# B&R Automation Studio project RS15_RX_30005_r00 (part 2)

#### A7_BasicCyclic.st - Cyclic code
```iecst
(********************************************************************
 * COPYRIGHT -- Microsoft
 ********************************************************************
 * Program: A7_Basic
 * File: A7_BasicCyclic.st
 * Author: pkiel
 * Created: July 13, 2011
 ********************************************************************
 * Implementation of program A7_Basic
 ********************************************************************)

PROGRAM _CYCLIC

	gA[7].UnitsPerInch := gA[7].AxisPeriod/gRecipeActive.Repeat;
  gA[7].InchPerDeg := gA[7].UnitsPerDeg / gA[7].UnitsPerInch ;
  IF (g_rNumbPliers <> 0.0) THEN
    gA[7].rPerim_In := g_rSizeDrum_mm/g_rNumbPliers/25.4 ;
    gA[7].rRSynNum := 4.0 / g_rNumbPliers ;
  END_IF ;
  gA[7].rRSynDen := 1.0 ;

	IF (gA[7].Ident<>0) THEN

	(************************ READ DRIVE STATUS *************************)
	(* Access to the following bools:
	gA[x]_DriveStatus.Simulation			: If TRUE, simulation mode is active
	gA[x]_DriveStatus.NetworkInit			: If TRUE, the network is initialized
	gA[x]_DriveStatus.HomeSwitch			: If TRUE, the digital reference switch input is active
	gA[x]_DriveStatus.PosHWSwitch			: If TRUE, the positive hardware end switch is active
	gA[x]_DriveStatus.NegHWSwitch			: If TRUE, the negative hardware end switch is active
	gA[x]_DriveStatus.Trigger1				: If TRUE, the first trigger input is active
	gA[x]_DriveStatus.Trigger2				: If TRUE, the second trigger input is active
	gA[x]_DriveStatus.DriveEnable			: If TRUE, the enable input is active
	gA[x]_DriveStatus.ControllerReady		: If TRUE, the controller is ready to beturned on
	gA[x]_DriveStatus.ControllerStatus		: If TRUE, the controller is turned on (Same as MC_Power.Status)
	gA[x]_DriveStatus.AxisError				: If TRUE, at least one error has occurred (not acknowledged)
	gA[x]_DriveStatus.LagWarning			: If TRUE, the lag error has exceeded the limit value specified for a warning*)
		MC_BR_ReadDriveStatus_0.Enable := 1;
		MC_BR_ReadDriveStatus_0.Axis := gA[7].Ident;
		MC_BR_ReadDriveStatus_0.AdrDriveStatus := ADR (DriveStatus);
		MC_BR_ReadDriveStatus_0();
		gA[7].Ind_Simulation		:=	DriveStatus.Simulation;
		gA[7].Ind_NetworkInit		:=	DriveStatus.NetworkInit;
		gA[7].Input_Home			:=	DriveStatus.HomeSwitch;
		gA[7].Input_PosHW			:=	DriveStatus.PosHWSwitch;
		gA[7].Input_NegHW			:=	DriveStatus.NegHWSwitch;
		gA[7].Input_Trigger1		:=	DriveStatus.Trigger1;
		gA[7].Input_Trigger2		:=	DriveStatus.Trigger2;
		gA[7].Input_DriveEnable		:=	DriveStatus.DriveEnable;
		gA[7].Ind_ControllerReady	:=	DriveStatus.ControllerReady;
		gA[7].Ind_ControllerStatus	:=	DriveStatus.ControllerStatus;
		gA[7].Error					:=	DriveStatus.AxisError;
		gA[7].Ind_LagWarning		:=	DriveStatus.LagWarning;

	(************************ READ AXIS ERROR **********************)
		MC_ReadAxisError_0.Enable := gA[7].Ind_NetworkInit;
		MC_ReadAxisError_0.Axis := gA[7].Ident;
		MC_ReadAxisError_0.DataAddress := ADR(gA[7].ErrorText);
		MC_ReadAxisError_0.DataLength := SIZEOF(gA[7].ErrorText);
		MC_ReadAxisError_0.DataObjectName := 'Error_Eng';
		MC_ReadAxisError_0();
		IF(MC_ReadAxisError_0.Valid) THEN
			gA[7].ErrorID := MC_ReadAxisError_0.AxisErrorID;
			gA[7].ErrorCount := MC_ReadAxisError_0.AxisErrorCount;
		END_IF
	(* Auto Acknowledge Errors *)
		IF (gA[7].Cmd_Reset AND (gA[7].ErrorCount<>0) AND NOT AutoAck) THEN
			AutoAck:=1;
		ELSE
			AutoAck:=0;
		END_IF
	(*Axis Error Acknowledge*)
		IF (EDGEPOS(AutoAck) OR EDGEPOS(gA[7].ErrorAck)) THEN
			MC_ReadAxisError_0.Acknowledge := 1;
		ELSE;
			MC_ReadAxisError_0.Acknowledge :=0;
		END_IF

	(************************ RESET AXIS ERROR **********************)
		IF (gA[7].Cmd_Reset AND (gA[7].ErrorCount=0) AND gA[7].ErrorStop) THEN
			MC_Reset_0.Execute:=1;
		END_IF
		IF (MC_Reset_0.Done) THEN
			MC_Reset_0.Execute:=0;
			gA[7].Cmd_Reset:=0;
			ResetError := 0;
		END_IF
		IF (MC_Reset_0.Error) THEN
			MC_Reset_0.Execute:=0;
			gA[7].Cmd_Reset:=0;
			ResetError := 1;
		END_IF
		MC_Reset_0.Axis:=gA[7].Ident;
		MC_Reset_0();

	(************************ READ AXIS STATUS *************************)
		MC_ReadStatus_0.Enable := gA[7].Ind_NetworkInit;
		MC_ReadStatus_0.Axis := gA[7].Ident;
		MC_ReadStatus_0();
		IF(MC_ReadStatus_0.Valid = TRUE)THEN
			gA[7].Ind_Enabled 			:= NOT (MC_ReadStatus_0.Disabled);
			gA[7].Ind_StandStill		:= MC_ReadStatus_0.StandStill;
			gA[7].Ind_Stopping			:= MC_ReadStatus_0.Stopping;
			gA[7].Ind_DiscreteMotion	:= MC_ReadStatus_0.DiscreteMotion;
			gA[7].Ind_ContinuousMotion	:= MC_ReadStatus_0.ContinuousMotion;
			gA[7].Ind_SynchronizedMotion:= MC_ReadStatus_0.SynchronizedMotion;
			gA[7].ErrorStop				:= MC_ReadStatus_0.Errorstop;
		END_IF
    IF NOT(gA[7].Ind_Enabled) THEN
      gA[7].bSynchroReq := 1 ;
    END_IF
    IF EDGEPOS(gA[7].Ind_bSynchroOK) THEN
      gA[7].bSynchroReq := 0 ;
    END_IF

	(******************** INIT POSITION MODULUS  *********************)
    IF (g_rNumbPliers <> 0.0) THEN
      IF ( gA[7].Ind_StandStill     OR
           NOT(gA[7].Ind_Enabled) ) AND
         g_bChangeModDrumReq        THEN
        bChangeModReq := 1 ;
        uiInitModPos0_ErrorID := 0 ;
      END_IF
      MC_BR_InitModPos_0.Execute:= (InitModPosition OR bChangeModReq) ;
  		MC_BR_InitModPos_0.Axis:= gA[7].Ident;
  		MC_BR_InitModPos_0.Period:= REAL_TO_UDINT(gA[7].AxisPeriod * 4.0/g_rNumbPliers);
  		MC_BR_InitModPos_0.Factor:=1;
  		InitModPos_Done:=MC_BR_InitModPos_0.Done;
    END_IF
    IF MC_BR_InitModPos_0.Done THEN
      g_bChangeModDrumReq := 0 ;
      bChangeModReq       := 0 ;
    ELSIF MC_BR_InitModPos_0.Error THEN
      bChangeModReq := 0 ;
      uiInitModPos0_ErrorID := MC_BR_InitModPos_0.ErrorID ;
    END_IF
		MC_BR_InitModPos_0();

	(******************** INIT ENDLESS POSITION *********************)
		MC_BR_InitEndlessPosition_0.Execute:= InitModPos_Done;
		MC_BR_InitEndlessPosition_0.Axis:= gA[7].Ident;
		MC_BR_InitEndlessPosition_0.DataAddress:= ADR(gEndPosData[7]);
		IF (MC_BR_InitEndlessPosition_0.Done) THEN
			InitModPosition:=0;
			InitEndlessPosition:=0;
			HomeRestore:=1;
		END_IF
		MC_BR_InitEndlessPosition_0();

	(************************ HOME AXIS FIRST POWER UP **********************)
		IF (HomeRestore AND NOT gA7_FirstHomed) THEN
			MC_Home_0.Execute:=1;
		END_IF
		MC_Home_0.Axis:=gA[7].Ident;
		MC_Home_0.Position:=0;
		MC_Home_0.HomingMode:=mcHOME_DIRECT;
		IF (MC_Home_0.Done) THEN
			MC_Home_0.Execute:=0;
			gA7_FirstHomed:=1;
		END_IF
		MC_Home_0();

	(************************ HOME AXIS **********************)
		IF (gA7_FirstHomed) THEN
			MC_Home_1.Execute:=HomeRestore;
		END_IF
		MC_Home_1.Axis:=gA[7].Ident;
		MC_Home_1.Position:=0;
		MC_Home_1.HomingMode:=mcHOME_RESTORE_POS;
		IF (MC_Home_1.Done) THEN
			gA[7].Ind_Homed:=1;
			HomeRestore:=0;
		END_IF
		MC_Home_1();

	(******************** READ ACTUAL POSITION *********************)
		MC_ReadActualPosition_0.Enable:= gA[7].Ind_NetworkInit;
		MC_ReadActualPosition_0.Axis:= gA[7].Ident;
		MC_ReadActualPosition_0();
		IF(MC_ReadActualPosition_0.Valid = TRUE)THEN
			gA[7].PositionCount := MC_ReadActualPosition_0.Position;
			gA[7].PositionInch := gA[7].PositionCount/gA[7].UnitsPerInch;
			gA[7].PositionDeg := gA[7].PositionCount/gA[7].UnitsPerDeg;
		END_IF

  //******************** READ SET POINT POSITION *********************
    // Slave side  : ParID 428 SGEN_S_SET : CTRL Position controller: Input set position
    // Master side : ParID 412 S_SET_VAX1 : 412: VAX: Position

    // Slave side
    MC_BR_CyclicRead_0.Axis        := gA[7].Ident ;
    MC_BR_CyclicRead_0.Enable      := gA[7].Ind_NetworkInit;
    MC_BR_CyclicRead_0.ParID       := 428 ;
    MC_BR_CyclicRead_0.DataAddress := ADR(iiSP_SlPos_U);
    MC_BR_CyclicRead_0.DataType    := ncPAR_TYP_DINT ;
    // Master side
    MC_BR_CyclicRead_1.Axis        := gA[9].Ident ;
    MC_BR_CyclicRead_1.Enable      := gA[7].Ind_NetworkInit;
    MC_BR_CyclicRead_1.ParID       := 412 ;
    MC_BR_CyclicRead_1.DataAddress := ADR(iiSP_MaPos_U);
    MC_BR_CyclicRead_1.DataType    := ncPAR_TYP_DINT ;

    IF MC_BR_CyclicRead_0.Valid THEN
      rSP_SlPos_Deg := iiSP_SlPos_U/gA[7].UnitsPerDeg ;
    ELSIF MC_BR_CyclicRead_0.Error THEN
      MC_BR_CyclicRead_0.Enable := 0 ;
    END_IF
    IF MC_BR_CyclicRead_1.Valid THEN
      rSP_MaPos_Deg := iiSP_MaPos_U/gA[9].UnitsPerDeg ;
    ELSIF MC_BR_CyclicRead_1.Error THEN
      MC_BR_CyclicRead_1.Enable := 0 ;
    END_IF
    MC_BR_CyclicRead_0();
    MC_BR_CyclicRead_1();

  //******************** READ ACTUAL OFFSET *********************
  IF gA[7].rRSynDen > 0.0 THEN
    rTempActPhasDeg := rSP_SlPos_Deg - gA[7].rRSynNum / gA[7].rRSynDen * rSP_MaPos_Deg ;
    gA[7].rActPhasDeg := H_FC_Modulus (
                              IN_rMod := 360 * gA[7].rRSynNum / gA[7].rRSynDen ,
                              IN_rVar := rTempActPhasDeg
                                      ) ;
  END_IF

	(******************** READ ACTUAL VELOCITY *********************)
		IF(MC_ReadActualVelocity_0.Error=TRUE) THEN
			MC_ReadActualVelocity_0.Enable:= 0;
		ELSE
			MC_ReadActualVelocity_0.Enable:= 1;
		END_IF
		MC_ReadActualVelocity_0.Axis:= gA[7].Ident;
		MC_ReadActualVelocity_0();
		IF(MC_ReadActualVelocity_0.Valid = TRUE)THEN
			//gA[7].ActualVelocity := MC_ReadActualVelocity_0.Velocity*60/gA[7].SP_MotorPPR;
      gA[7].ActualVelocity := MC_ReadActualVelocity_0.Velocity*60/gA[7].AxisPeriod ; // D.M. 03/08/2011 BrownPaper_14542  Need speed of the axis and not of the shaft of the motor
      IF ABS(gA[7].ActualVelocity>1) THEN // D.M. 03/08/2011 BrownPaper_14542 Add ABS because in case negative velocity Ind_InMotion = 0 instead of 1
				gA[7].Ind_InMotion:=1;
			ELSE
				gA[7].Ind_InMotion:=0;
			END_IF
		END_IF

	(******************** READ ACTUAL TORQUE *********************)
		IF(MC_ReadActualTorque_0.Error=TRUE) THEN
			MC_ReadActualTorque_0.Enable:= 0;
		ELSE
			MC_ReadActualTorque_0.Enable:= 1;
		END_IF
		MC_ReadActualTorque_0.Axis:= gA[7].Ident;
		MC_ReadActualTorque_0();
		IF(MC_ReadActualTorque_0.Valid = TRUE)THEN
			gA[7].ActualTorque := MC_ReadActualTorque_0.Torque;
		END_IF

	(************************ ENABLE AXIS **********************)
		MC_Power_0.Axis:=gA[7].Ident;
		IF (MC_Power_0.Error=0) THEN
			MC_Power_0.Enable:=gA[7].Cmd_Enable;
		ELSE;
			MC_Power_0.Enable:=0;
		END_IF;
		MC_Power_0();

	(************************ AXIS VELOCITY MOVE **********************)
		MC_MoveVelocity_0.Axis:=gA[7].Ident;
		MC_MoveVelocity_0.Velocity:=gA[7].SP_Velocity*gA[7].AxisPeriod/60;
		MC_MoveVelocity_0.Acceleration:=gA[7].SP_Accel;
		MC_MoveVelocity_0.Deceleration:=gA[7].SP_Decel;
		MC_MoveVelocity_0.Direction:=mcPOSITIVE_DIR;
		IF ((EDGEPOS(gA[7].Cmd_ContinuousMotion)) OR (EDGEPOS(gA[7].Cmd_ContinuousMotionUpdate))) THEN
			MC_MoveVelocity_0.Execute:=1;
		ELSE
			MC_MoveVelocity_0.Execute:=0;
		END_IF;
		MC_MoveVelocity_0();

  //************************ AXIS OVERRIDE **********************
    MC_SetOverride_0.Axis      := gA[7].Ident ;
    MC_SetOverride_0.Enable    := gA[7].Cmd_Override ;
    MC_SetOverride_0.VelFactor := gA[7].rSP_OverrideV ;
    MC_SetOverride_0.AccFactor := gA[7].rSP_OverrideA ;
    IF (MC_SetOverride_0.Enabled) OR
       (MC_SetOverride_0.Error)   THEN
      gA[7].Cmd_Override := 0 ;
    END_IF
    MC_SetOverride_0();

	(************************ AXIS STOP **********************)
		MC_Stop_0.Axis:=gA[7].Ident;
		IF (gA[7].Ind_ContinuousMotion AND (NOT gA[7].Cmd_ContinuousMotion) AND gAlarmsOK) THEN
			MC_Stop_0.Deceleration:=gA[7].SP_Decel;
			MC_Stop_0.Execute:=1;
		END_IF;
		IF (MC_Stop_0.Done OR MC_Stop_0.CommandAborted OR MC_Stop_0.Error) THEN
			MC_Stop_0.Execute:=0;
		END_IF;
		MC_Stop_0();

  (************************  ESTOP **********************)
    MC_Stop_1.Axis:=gA[7].Ident;
    IF EDGEPOS(g_bIndEStopStandstill) THEN
      MC_Stop_1.Deceleration:=gA[7].SP_EStopDecel;
      MC_Stop_1.Execute:=1;
    END_IF;
    IF (MC_Stop_1.Done OR MC_Stop_1.CommandAborted OR MC_Stop_1.Error) THEN
      MC_Stop_1.Execute:=0;
      gA[7].Cmd_EStopDisable := 1 ;
    END_IF;
    IF NOT(g_bIndEStopStandstill) THEN
      gA[7].Cmd_EStopDisable := 0 ;
    END_IF;
    MC_Stop_1();

    //************************ AXIS PHASE CONTROL (Inches) First Step **********************
    IF EDGEPOS(gA[7].Cmd_PhaseOffset) THEN
      rSP_PhaseOffsetVal := gA[7].SP_PhaseOffset ;
    END_IF;

    (************************ SHIFTING PERF CONTROL **********************)
    IF g_bCmdShiftA[7] THEN
      //rSP_ShiftDrum := g_iPerfShiftPos * gr_rIncrShiftPerf_mm/25.4 * gA[7].rRSynNum/gA[7].rRSynDen ;  // D.M. RS26_Pyrollpack_14661 CAUTION !!! Phasing acts on the master side and not slave side, replaced by the code below
      rSP_ShiftDrum := g_iPerfShiftPos * gr_rIncrShiftPerf_mm/25.4 ;
      gA[7].Cmd_PhaseOffset := 1 ;
      g_bCmdShiftA[7] := 0 ;
    END_IF

    (************************ AXIS PHASE CONTROL (Inches) Next Step **********************)
    // The biggers Offsets are divided in several successives shifts to not damage the blades on the Drum du to too much acceleration
    IF gA[7].Cmd_PhaseOffset               AND
       ( EDGENEG(gA[7].Ind_bInContactZone) AND
         (g_iMachType <> C_iRS15)          OR
         EDGENEG(gA[4].Ind_bInContactZone) AND
         (g_iMachType = C_iRS15) )         THEN
      gA[7].Cmd_PhaseOffset := 0 ;
      rSP_PhaseOffset := rSP_PhaseOffsetVal + rSP_ShiftDrum ;
      bCmd_PhaseOffset := 1 ;
      g_bIndPhasDrumInact := 0 ;
      //iTest_[0] := 0 ;
      //iTest_[1] := 0 ;
      //iTest_[2] := 0 ;
      //iTest_[3] := 0 ;
    END_IF
    rMaxShift := gr_rLimOffsetRunVal * gRecipeActive.Repeat ;
    // Signe of the Offset
    IF (rSP_PhaseOffset <> 0.0) THEN
      rShiftSign := rSP_PhaseOffset / ABS(rSP_PhaseOffset) ;
    END_IF
    // Shift calculation
    IF bCmd_PhaseOffset THEN
      IF (ABS(rSP_PhaseOffset) > rMaxShift) THEN
        rSP_ShiftVal := rMaxShift * rShiftSign ;
        rSP_PhaseOffset := rSP_PhaseOffset - rSP_ShiftVal ;
        iTest_[0] := iTest_[0] + 1 ;
      ELSE
        rSP_ShiftVal := rSP_PhaseOffset ;
        rSP_PhaseOffset := 0.0 ;
        iTest_[1] := iTest_[1] + 1 ;
      END_IF
    END_IF

    MC_BR_Phasing_0.Slave:=gA[7].Ident;
    IF gA[7].Ind_SynchronizedMotion AND NOT(gstCycA[7].CycManTimSet.bSCyc) AND st_TON_0.Q THEN
      MC_BR_Phasing_0.Enable:= 1;
    ELSE;
      MC_BR_Phasing_0.Enable:=0;
    END_IF;
    IF bCmd_PhaseOffset AND NOT(gstCycA[7].CycManTimSet.bSCyc) THEN
      MC_BR_Phasing_0.InitData:=1;
      bCmd_PhaseOffset := 0 ;
      IF (rSP_PhaseOffset = 0.0) THEN
        // Calculation new phase Drum/Master
        rTemp_[4] := (rSP_PhaseOffsetVal+rSP_ShiftDrum)/gA[7].InchPerDeg ;
        rTemp_[5] := gRecipeActive.rDrum_PhasMasterDeg + rTemp_[4]*gA[7].rRSynNum/gA[7].rRSynDen ;
        gRecipeActive.rDrum_PhasMasterDeg := H_FC_Modulus (IN_rMod := 360*gA[7].rRSynNum/gA[7].rRSynDen, IN_rVar := rTemp_[5]) ;
        rSP_ShiftDrum := 0.0 ;
        rSP_PhaseOffsetVal := 0 ;
        iTest_[2] := iTest_[2] + 1 ;
      END_IF;
    ELSE
      MC_BR_Phasing_0.InitData:=0;
    END_IF
    MC_BR_Phasing_0.Shift               := rSP_ShiftVal*gA[9].UnitsPerInch;
    MC_BR_Phasing_0.Velocity            := 6*gA[7].AxisPeriod/60;
    MC_BR_Phasing_0.Acceleration        := gA[7].SP_Decel;
    MC_BR_Phasing_0.ApplicationDistance := 0.8*gA[9].AxisPeriod * gA[7].rRSynNum/gA[7].rRSynDen ;
    MC_BR_Phasing_0.ApplicationMode     := mcMASTER_DISTANCE_BASED;
    MC_BR_Phasing_0.ShiftMode           := mcRELATIVE;
    MC_BR_Phasing_0();

    IF MC_BR_Phasing_0.ShiftAttained       AND
       (rSP_PhaseOffset <> 0.0)            AND
       ( EDGENEG(gA[7].Ind_bInContactZone) AND
         (g_iMachType <> C_iRS15)          OR
         EDGENEG(gA[4].Ind_bInContactZone) AND
         (g_iMachType = C_iRS15) )         THEN
      bCmd_PhaseOffset := 1 ;
      iTest_[3] := iTest_[3] + 1 ;
    END_IF
    // Drum phasing inactive
    IF (rSP_PhaseOffset=0.0)         AND
       MC_BR_Phasing_0.ShiftAttained OR
       NOT(MC_BR_Phasing_0.Busy)     AND
       1                             THEN
      g_bIndPhasDrumInact := 1 ;
    END_IF

    (************************ AXIS PHASE CONTROL (Inches) TIMING SETTING **********************)
    IF gstCycA[7].CycManTimSet.bSCyc THEN
      IF gA[7].Cmd_ManuTimSetPlus THEN
        rAxisTimSet_SP_Vel := gr_rAxisTimSet_SP_Vel*gA[9].AxisPeriod/60 / (gA[7].rRSynNum/gA[7].rRSynDen) ;
      ELSE
        rAxisTimSet_SP_Vel := - gr_rAxisTimSet_SP_Vel*gA[9].AxisPeriod/60 / (gA[7].rRSynNum/gA[7].rRSynDen) ;
      END_IF
        rAxisTimSet_SP_Acc := gr_rAxisTimSet_SP_Acc*gA[9].AxisPeriod/60/60 ;
    END_IF

    MC_BR_Phasing_1.Slave                  := gA[7].Ident;
    MC_BR_Phasing_1.Enable                 := gstCycA[7].CycManTimSet.bCyc ;
    MC_BR_Phasing_1.InitData               := gstCycA[7].CycManTimSet.bSCyc ;
    MC_BR_Phasing_1.PerformVelocityControl := gstCycA[7].CycManTimSet.CmdMov ;
    MC_BR_Phasing_1.Velocity               := rAxisTimSet_SP_Vel ;
    MC_BR_Phasing_1.Acceleration           := rAxisTimSet_SP_Acc ;
    MC_BR_Phasing_1.ApplicationMode        := mcVELOCITY_CONTROL ;
    MC_BR_Phasing_1();
    st_TON_0(IN:=NOT(MC_BR_Phasing_1.Enable),PT:=T#100ms) ;

    IF NOT(gstCycA[7].CycManTimSet.CmdMov) AND
       MC_BR_Phasing_1.ShiftAttained       OR
       NOT(gstCycA[7].CycManTimSet.bCyc)   OR
       MC_BR_Phasing_1.Error               AND
       1                                   THEN
      gstCycA[7].CycManTimSet.CmdStop := 0 ;
    END_IF
	END_IF

END_PROGRAM
```

#### A7_Basic.var - Local variables
```iecst
(********************************************************************
 * COPYRIGHT -- Microsoft
 ********************************************************************
 * Program: A7_Basic
 * File: A7_Basic.var
 * Author: pkiel
 * Created: July 13, 2011
 ********************************************************************
 * Local variables of program A7_Basic
 ********************************************************************)
VAR
	AutoAck : BOOL;
	AxisErrorNcAccess : UINT;
	DriveStatus : MC_DRIVESTATUS_TYP;
	HomeRestore : BOOL;
	InitEndlessPosition : BOOL;
	InitModPos_Done : BOOL;
	InitModPosition : BOOL;
	MC_BR_InitEndlessPosition_0 : MC_BR_InitEndlessPosition;
	MC_BR_InitModPos_0 : MC_BR_InitModPos;
  uiInitModPos0_ErrorID : UINT ;
  MC_BR_Phasing_0 : MC_BR_Phasing;
  rSP_PhaseOffset  : REAL ;
  rSP_ShiftVal     : REAL ;
  rShiftSign       : REAL ;
  rMaxShift        : REAL ;
  bCmd_PhaseOffset : BOOL ;
  MC_BR_Phasing_1 : MC_BR_Phasing;
	MC_BR_ReadDriveStatus_0 : MC_BR_ReadDriveStatus;
	MC_Home_0 : MC_Home;
	MC_Home_1 : MC_Home;
	MC_MoveVelocity_0 : MC_MoveVelocity;
	MC_Power_0 : MC_Power;
	MC_ReadActualPosition_0 : MC_ReadActualPosition;
	MC_ReadActualTorque_0 : MC_ReadActualTorque;
	MC_ReadActualVelocity_0 : MC_ReadActualVelocity;
	MC_ReadAxisError_0 : MC_ReadAxisError;
	MC_ReadStatus_0 : MC_ReadStatus;
	MC_Reset_0 : MC_Reset;
  MC_Stop_0 : MC_Stop;
  MC_Stop_1 : MC_Stop;
  st_TON_0 : TON ;
	ResetError : BOOL;
  rTemp_ : ARRAY[0..9] OF REAL ;
  bTest_ : ARRAY[0..9] OF BOOL ;
  rTest_ : ARRAY[0..9] OF REAL ;
  iTest_ : ARRAY[0..9] OF INT ;
  rAxisTimSet_SP_Vel  : REAL ; (*Set point Velocity for Axis manual timing setting cycle, in units/s*)
  rAxisTimSet_SP_Acc  : REAL ; (*Set point Acceleration for Axis manual timing setting cycle, in units/s²*)
  rAxisTimSet_SP_Dec  : REAL ; (*Set point Deceleration for Axis manual timing setting cycle, in units/s²*)
  uiAxisTimSet_SP_Dir : USINT ; (*Set point Direction for Axis manual timing setting cycle*)
  uiAxisTimSet_SP_ShiftAppMode : UINT ; (*Set point Shit Application mode for phasing Axis manual timing setting cycle*)
  rTempActPhasDeg : REAL;
  rA9PosCorDeg  : REAL;
  rRepeatMetric : REAL;
  MC_SetOverride_0 : MC_SetOverride;

  iiSP_SlPos_U  : DINT ; (*On Slave side, input set point position of the position controller ParID 428, in unit*)
  rSP_SlPos_Deg : REAL ; (*On Slave side, input set point position of the position controller ParID 428, in deg*)
  iiSP_MaPos_U  : DINT ; (*On Master side, input set point position of the position controller ParID 412, in unit*)
  rSP_MaPos_Deg : REAL ; (*On Master side, input set point position of the position controller ParID 412, in deg*)
  MC_BR_CyclicRead_0 : MC_BR_CyclicRead ;
  MC_BR_CyclicRead_1 : MC_BR_CyclicRead ;

  bChangeModReq      : BOOL ;
  uiOffsetStat       : UINT ;
  rSP_ShiftDrum      : REAL ;
  SP_PhaseOffset     : REAL ;
  rSP_PhaseOffsetVal : REAL ;
END_VAR
```

### Program Logical/BagMachine_Section/Drum/Axis7/A7_Control (IEC) - Servo Control

#### A7_Control.var
```iecst
(********************************************************************
 * COPYRIGHT -- Microsoft
 ********************************************************************
 * Program: A7_Control
 * File: A7_Control.var
 * Author: pkiel
 * Created: July 13, 2011
 ********************************************************************
 * Local variables of program A7_Control
 ********************************************************************)
VAR
	HGW_ChangeReal_0 : HGW_ChangeReal;
	HGW_RelativeChangeReal_0 : H_FB_RelativeChangeLimitReal1;
	HGW_Toggle_0 : HGW_Toggle;
	Synch_Permissive : BOOL;
	TOF_0 : TOF;
	TON_0 : TON;
  rIncrOffsetAxeRun_Inch : REAL ;
END_VAR
```

#### A7_ControlCyclic.ld
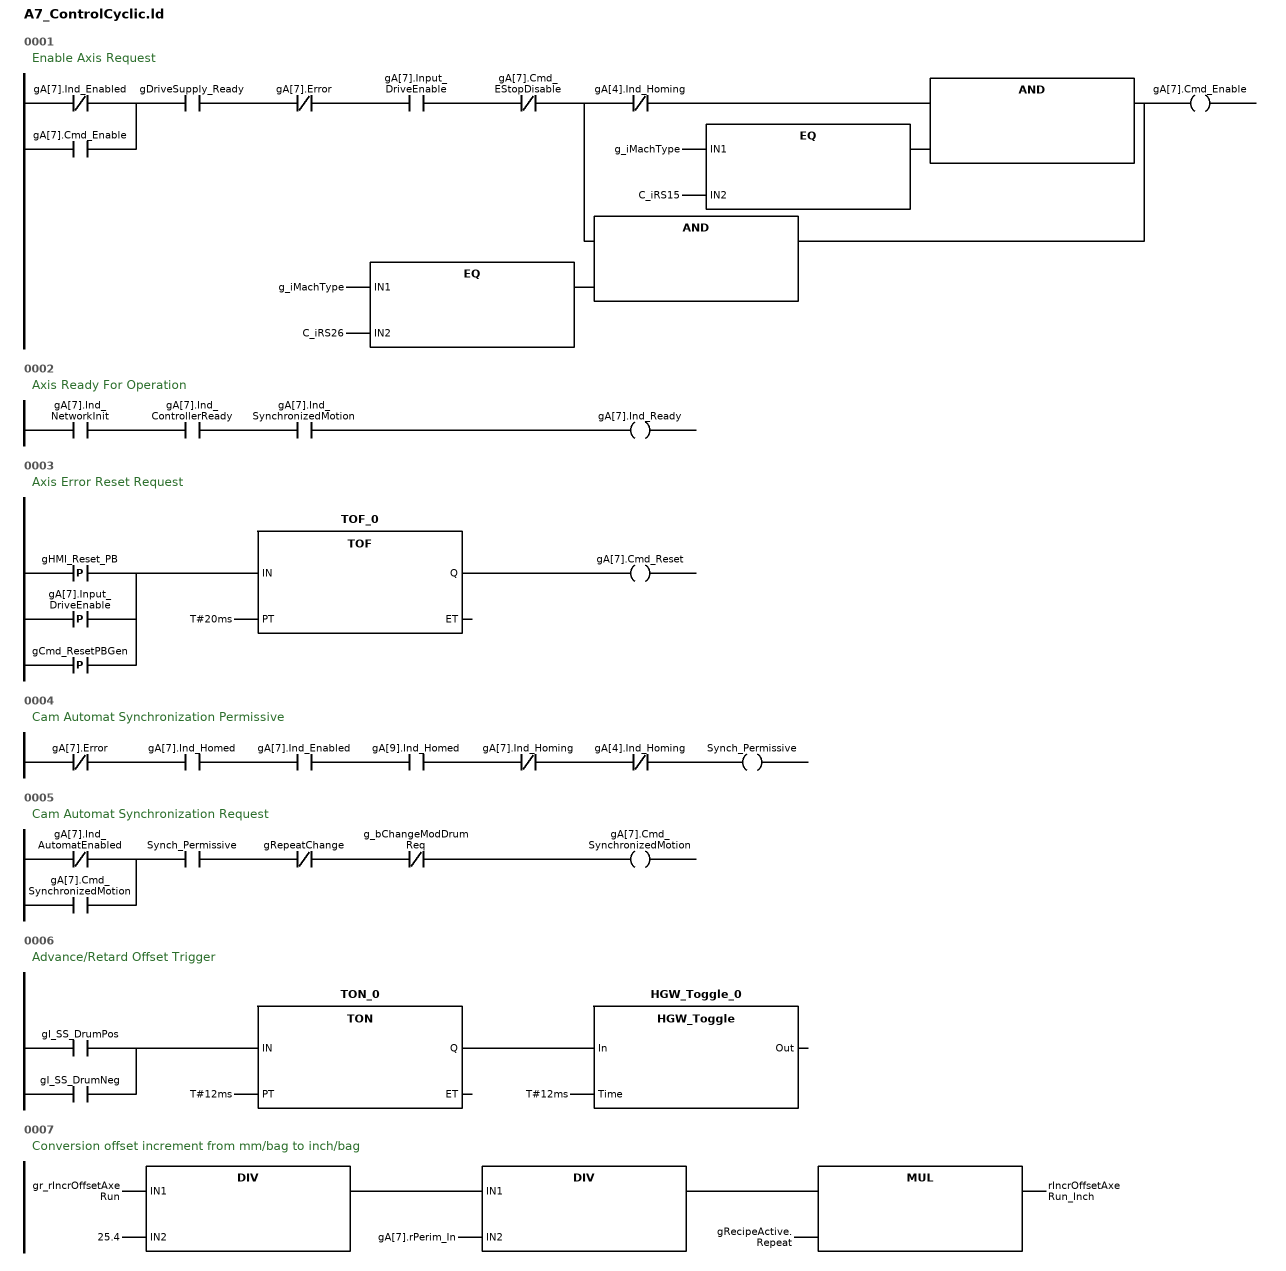
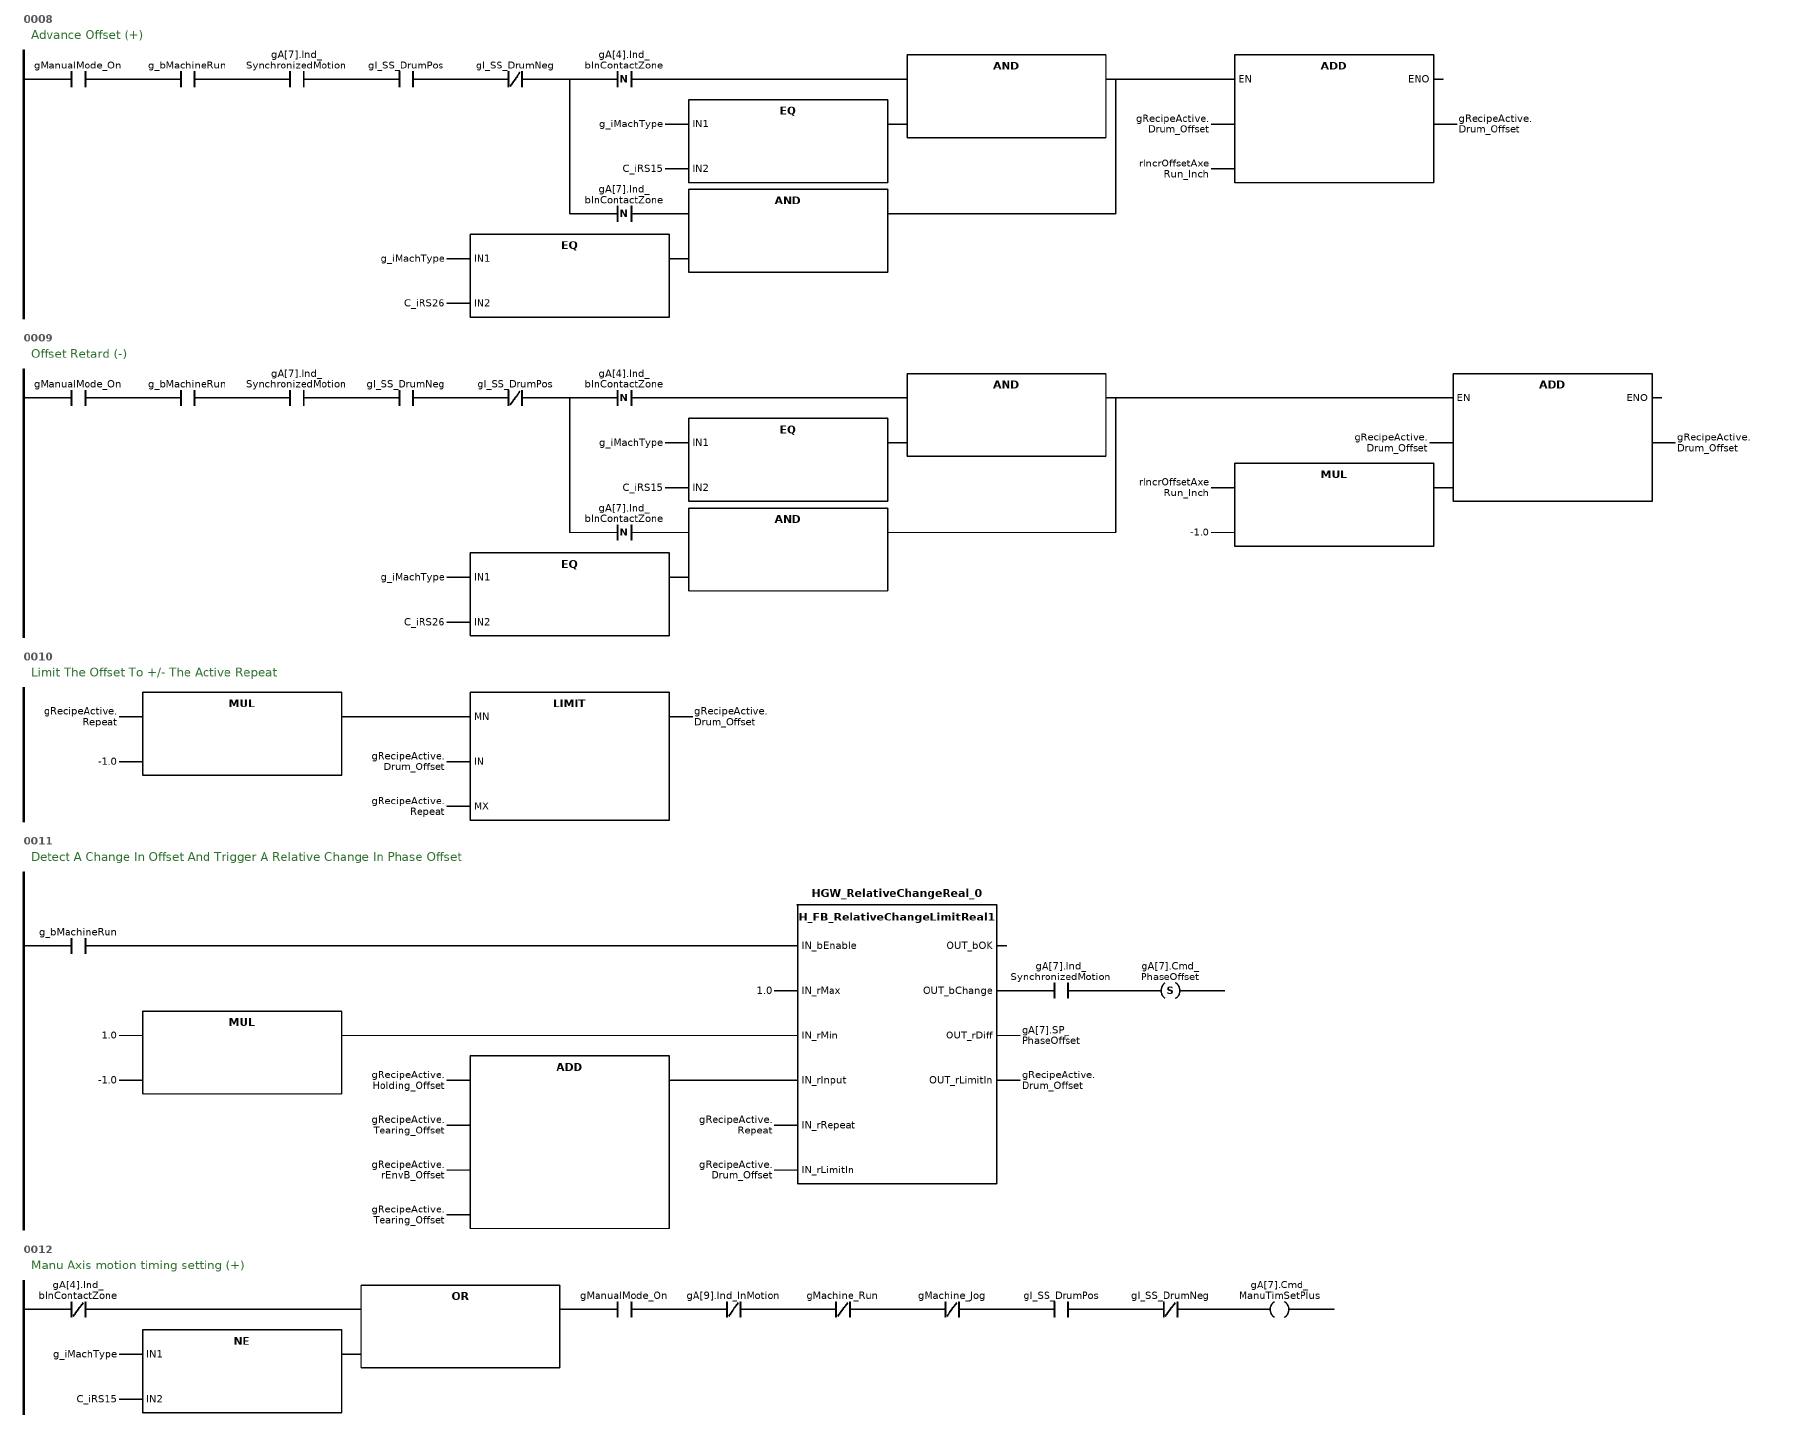
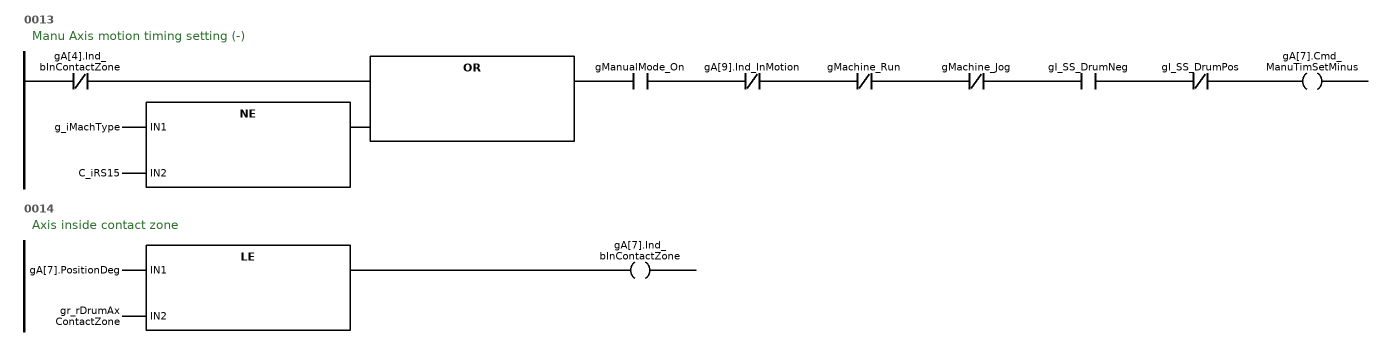
Ladder, written as Structured Text:
```iecst
(********************************************************************
 * COPYRIGHT -- Microsoft
 ********************************************************************
 * Program: A7_Control
 * File: A7_ControlCyclic.ld
 * Author: pkiel
 * Created: July 13, 2011
 ********************************************************************
 * Implementation of program A7_Control
 ********************************************************************)

PROGRAM _CYCLIC
VAR
    _p1 : BOOL;
    _e2 : R_TRIG;
    _e3 : R_TRIG;
    _e4 : R_TRIG;
    _p5 : BOOL;
    _e6 : F_TRIG;
    _e7 : F_TRIG;
    _p8 : BOOL;
    _e9 : F_TRIG;
    _e10 : F_TRIG;
END_VAR
(* Network 1: Enable Axis Request *)
_p1 := (NOT gA[7].Ind_Enabled OR gA[7].Cmd_Enable) AND gDriveSupply_Ready AND NOT gA[7].Error AND gA[7].Input_DriveEnable AND NOT gA[7].Cmd_EStopDisable;
gA[7].Cmd_Enable := _p1 AND ((NOT gA[4].Ind_Homing AND (g_iMachType = C_iRS15)) OR (g_iMachType = C_iRS26));

(* Network 2: Axis Ready For Operation *)
gA[7].Ind_Ready := gA[7].Ind_NetworkInit AND gA[7].Ind_ControllerReady AND gA[7].Ind_SynchronizedMotion;

(* Network 3: Axis Error Reset Request *)
_e2(CLK := gHMI_Reset_PB);
_e3(CLK := gA[7].Input_DriveEnable);
_e4(CLK := gCmd_ResetPBGen);
TOF_0(IN := _e2.Q OR _e3.Q OR _e4.Q, PT := T#20ms);
gA[7].Cmd_Reset := TOF_0.Q;

(* Network 4: Cam Automat Synchronization Permissive *)
Synch_Permissive := NOT gA[7].Error AND gA[7].Ind_Homed AND gA[7].Ind_Enabled AND gA[9].Ind_Homed AND NOT gA[7].Ind_Homing AND NOT gA[4].Ind_Homing;

(* Network 5: Cam Automat Synchronization Request *)
gA[7].Cmd_SynchronizedMotion := (NOT gA[7].Ind_AutomatEnabled OR gA[7].Cmd_SynchronizedMotion) AND Synch_Permissive AND NOT gRepeatChange AND NOT g_bChangeModDrumReq;

(* Network 6: Advance/Retard Offset Trigger *)
TON_0(IN := gI_SS_DrumPos OR gI_SS_DrumNeg, PT := T#12ms);
HGW_Toggle_0(In := TON_0.Q, Time := T#12ms);

(* Network 7: Conversion offset increment from mm/bag to inch/bag *)
rIncrOffsetAxeRun_Inch := ((gr_rIncrOffsetAxeRun / 25.4) / gA[7].rPerim_In) * gRecipeActive.Repeat;

(* Network 8: Advance Offset (+) *)
_p5 := gManualMode_On AND g_bMachineRun AND gA[7].Ind_SynchronizedMotion AND gI_SS_DrumPos AND NOT gI_SS_DrumNeg;
_e6(CLK := gA[4].Ind_bInContactZone);
_e7(CLK := gA[7].Ind_bInContactZone);
IF _p5 AND ((_e6.Q AND (g_iMachType = C_iRS15)) OR (_e7.Q AND (g_iMachType = C_iRS26))) THEN
    gRecipeActive.Drum_Offset := gRecipeActive.Drum_Offset + rIncrOffsetAxeRun_Inch;
END_IF;

(* Network 9: Offset Retard (-) *)
_p8 := gManualMode_On AND g_bMachineRun AND gA[7].Ind_SynchronizedMotion AND gI_SS_DrumNeg AND NOT gI_SS_DrumPos;
_e9(CLK := gA[4].Ind_bInContactZone);
_e10(CLK := gA[7].Ind_bInContactZone);
IF _p8 AND ((_e9.Q AND (g_iMachType = C_iRS15)) OR (_e10.Q AND (g_iMachType = C_iRS26))) THEN
    gRecipeActive.Drum_Offset := gRecipeActive.Drum_Offset + (rIncrOffsetAxeRun_Inch * -1.0);
END_IF;

(* Network 10: Limit The Offset To +/- The Active Repeat *)
gRecipeActive.Drum_Offset := LIMIT(MN := gRecipeActive.Repeat * -1.0, IN := gRecipeActive.Drum_Offset, MX := gRecipeActive.Repeat);

(* Network 11: Detect A Change In Offset And Trigger A Relative Change In Phase Offset *)
HGW_RelativeChangeReal_0(IN_bEnable := g_bMachineRun, IN_rMax := 1.0, IN_rMin := 1.0 * -1.0, IN_rInput := gRecipeActive.Holding_Offset + gRecipeActive.Tearing_Offset + gRecipeActive.rEnvB_Offset + gRecipeActive.Tearing_Offset, IN_rRepeat := gRecipeActive.Repeat, IN_rLimitIn := gRecipeActive.Drum_Offset);
IF HGW_RelativeChangeReal_0.OUT_bChange AND gA[7].Ind_SynchronizedMotion THEN
    gA[7].Cmd_PhaseOffset := TRUE;
END_IF;
gA[7].SP_PhaseOffset := HGW_RelativeChangeReal_0.OUT_rDiff;
gRecipeActive.Drum_Offset := HGW_RelativeChangeReal_0.OUT_rLimitIn;

(* Network 12: Manu Axis motion timing setting (+) *)
gA[7].Cmd_ManuTimSetPlus := (NOT gA[4].Ind_bInContactZone OR (g_iMachType <> C_iRS15)) AND gManualMode_On AND NOT gA[9].Ind_InMotion AND NOT gMachine_Run AND NOT gMachine_Jog AND gI_SS_DrumPos AND NOT gI_SS_DrumNeg;

(* Network 13: Manu Axis motion timing setting (-) *)
gA[7].Cmd_ManuTimSetMinus := (NOT gA[4].Ind_bInContactZone OR (g_iMachType <> C_iRS15)) AND gManualMode_On AND NOT gA[9].Ind_InMotion AND NOT gMachine_Run AND NOT gMachine_Jog AND gI_SS_DrumNeg AND NOT gI_SS_DrumPos;

(* Network 14: Axis inside contact zone *)
gA[7].Ind_bInContactZone := gA[7].PositionDeg <= gr_rDrumAxContactZone;
END_PROGRAM
```

### Program Logical/BagMachine_Section/Drum/Axis7/A7_Automat (IEC) - Cam Automat

#### A7_AutomatCyclic.st
```iecst
(********************************************************************
 * COPYRIGHT -- Microsoft
 ********************************************************************
 * Program: A7_Automat
 * File: A7_AutomatCyclic.st
 * Author: pkiel
 * Created: July 13, 2011
 ********************************************************************
 * Implementation of program A7_Automat
 ********************************************************************)

PROGRAM _CYCLIC

(**** STRAIGHT GEARED CAM AUTOMAT WITH ABSOLUTE PHASE SYNCHRONIZATION FOR DRUM ***)

  // Set Up Master Position Parameter ID
  IF gstCycA[3].CycManTimSet.CmdSynchroOn  OR
     gstCycA[4].CycManTimSet.CmdSynchroOn  OR
     gstCycA[12].CycManTimSet.CmdSynchroOn OR
     gstCycA[13].CycManTimSet.CmdSynchroOn THEN
    MC_BR_AutControl_0.Signal1 := 1 ;
    MC_BR_AutControl_0.Signal2 := 0 ;
  ELSE
    MC_BR_AutControl_0.Signal1 := 0 ;
    MC_BR_AutControl_0.Signal2 := 1 ;
  END_IF

  // Select Master
  IF gA[12].bInMach             AND
     NOT(gA[13].bInMach)        AND
     gRecipeActive.bSelEnvBProd THEN
    uiiMaster := gA[12].Ident ;  // Case Envelope Bag One Axis
  END_IF
  IF gA[13].bInMach THEN
    uiiMaster := gA[13].Ident ;  // Case Envelope Bag Two Axis
  END_IF
  IF NOT(gA[12].bInMach) THEN
    uiiMaster := gA[4].Ident ;   // Case without Envelope Bag
  END_IF ;

  // Synchro OK indicator
  gstCycA[3].CycManTimSet.bSynchroOkSlavA[7] := ( MC_BR_InitMasterParIDTransfer_1.Master = uiiMaster )                                  AND
                                                ( MC_BR_InitMasterParIDTransfer_1.MasterParID = gstCycA[3].CycManTimSet.uiMasterParID ) AND
                                                ( MC_BR_AutControl_0.ActualStateIndex = 4 )                                             AND
                                                gA[7].Ind_SynchronizedMotion AND ParID_Ready ;

  gstCycA[4].CycManTimSet.bSynchroOkSlavA[7] := gstCycA[3].CycManTimSet.bSynchroOkSlavA[7] ;

  gstCycA[12].CycManTimSet.bSynchroOkSlavA[7] := ( MC_BR_InitMasterParIDTransfer_1.Master = uiiMaster )                                  AND
                                                ( MC_BR_InitMasterParIDTransfer_1.MasterParID = gstCycA[12].CycManTimSet.uiMasterParID ) AND
                                                ( MC_BR_AutControl_0.ActualStateIndex = 4 )                                              AND
                                                gA[7].Ind_SynchronizedMotion AND ParID_Ready ;

  gstCycA[13].CycManTimSet.bSynchroOkSlavA[7] := ( MC_BR_InitMasterParIDTransfer_1.Master = uiiMaster )                                  AND
                                                ( MC_BR_InitMasterParIDTransfer_1.MasterParID = gstCycA[13].CycManTimSet.uiMasterParID ) AND
                                                ( MC_BR_AutControl_0.ActualStateIndex = 4 )                                              AND
                                                gA[7].Ind_SynchronizedMotion AND ParID_Ready ;

  // Drum timing setting
  IF gstCycA[7].CycManTimSet.bCyc THEN
    IF gstCycA[7].CycManTimSet.CmdSynchroOn THEN
      MC_BR_AutControl_0.Signal1 := 1 ;
      MC_BR_AutControl_0.Signal2 := 0 ;
    ELSE
      MC_BR_AutControl_0.Signal1 := 0 ;
      MC_BR_AutControl_0.Signal2 := 1 ;
    END_IF
  END_IF

  IF gstCycA[3].CycManTimSet.bFCyc  AND
     gstCycA[4].CycManTimSet.bFCyc  AND
     gstCycA[7].CycManTimSet.bFCyc  AND
     gstCycA[12].CycManTimSet.bFCyc AND
     gstCycA[13].CycManTimSet.bFCyc THEN
    MC_BR_AutControl_0.Signal1 := 0 ;
    MC_BR_AutControl_0.Signal2 := 0 ;
  END_IF

  gstCycA[7].CycManTimSet.bSynchroOkSlavA[7] := ( MC_BR_AutControl_0.ActualStateIndex = 4 )  AND
                                                gA[7].Ind_SynchronizedMotion AND ParID_Ready ;

  //Synch_Request := gA[7].Cmd_SynchronizedMotion ;
  Synch_Request := gA[7].Cmd_SynchronizedMotion AND NOT(MC_BR_AutControl_0.Stop) ;  // D.M. 26/01/2012 RS26 Pyrollpack_14661 added because it happened that Stop=1 and Synch_Request=1 => MC_BR_AutControl_0 makes fault 29256
	IF (Synch_Request AND NOT ParID_Ready) THEN
	  MC_BR_InitMasterParIDTransfer_0.Master:= gA[9].Ident ;
    MC_BR_InitMasterParIDTransfer_0.Slave:= gA[7].Ident ;
    MC_BR_InitMasterParIDTransfer_0.MasterParID:= 412 ; // ParID 412 = 412: VAX: Position (in case virtual axis)
    MC_BR_InitMasterParIDTransfer_0.SlaveChannel:=0;
    MC_BR_InitMasterParIDTransfer_0.Execute:=TRUE;
    IF (MC_BR_InitMasterParIDTransfer_0.Done) THEN
      MasterParID:=MC_BR_InitMasterParIDTransfer_0.ReceiveParID;
      MC_BR_InitMasterParIDTransfer_0.Execute:=FALSE;
      ParID_Ready1:=1;
    ELSIF (MC_BR_InitMasterParIDTransfer_0.Error) THEN
    (*Store ErrorID in a variable,
      ErrorID is reset on falling edge of 'Execute'*)
      ErrorID:=MC_BR_InitMasterParIDTransfer_0.ErrorID;
      ParID_Ready1:=0;
      MC_BR_InitMasterParIDTransfer_0.Execute:=FALSE;
    END_IF
    MC_BR_InitMasterParIDTransfer_1.Master       := uiiMaster ;
    MC_BR_InitMasterParIDTransfer_1.Slave        := gA[7].Ident ;
    MC_BR_InitMasterParIDTransfer_1.MasterParID  := gstCycA[7].CycManTimSet.uiMasterParID ;
    MC_BR_InitMasterParIDTransfer_1.SlaveChannel := 5 ;
    MC_BR_InitMasterParIDTransfer_1.Execute      := TRUE ;
    IF (MC_BR_InitMasterParIDTransfer_1.Done) AND ParID_Ready1 THEN
      uiMasterParID1:=MC_BR_InitMasterParIDTransfer_1.ReceiveParID;
      MC_BR_InitMasterParIDTransfer_1.Execute:=FALSE;
      ParID_Ready:=1;
    ELSIF (MC_BR_InitMasterParIDTransfer_1.Error) THEN
    (*Store ErrorID in a variable,
      ErrorID is reset on falling edge of 'Execute'*)
      ErrorID:=MC_BR_InitMasterParIDTransfer_1.ErrorID;
      ParID_Ready:=0;
      MC_BR_InitMasterParIDTransfer_1.Execute:=FALSE;
    END_IF
	END_IF
  MC_BR_InitMasterParIDTransfer_0();
  MC_BR_InitMasterParIDTransfer_1();

(**** Initialize Automat Parameters Upon Automat Start Request ****)
	IF (EDGEPOS(ParID_Ready))THEN

		(**** Calculate Slave Start Offset ****)
      MasterOffset := gRecipeActive.Drum_Offset + gRecipeActive.Holding_Offset + gRecipeActive.Tearing_Offset;
			PositionOffset:= REAL_TO_DINT((gA[9].PositionInch-(gA[7].PositionInch-MasterOffset))*1000);
			PositionMOD:= REAL_TO_DINT(gRecipeActive.Repeat*1000);
			SlaveStartOffset:= (DINT_TO_REAL(PositionOffset MOD PositionMOD))/1000;
			IF (SlaveStartOffset >= (0.5*gRecipeActive.Repeat)) THEN
				SlaveStartOffset := SlaveStartOffset - gRecipeActive.Repeat;
			END_IF
			IF (SlaveStartOffset < (-0.5*gRecipeActive.Repeat)) THEN
				SlaveStartOffset := SlaveStartOffset + gRecipeActive.Repeat;
      END_IF

		(*general automat parameter*)
			(*AutData.Master			  	:= gA1.Ident;*)
			AutData.MasterParID	  		:= MasterParID;
			AutData.StartPosition  		:= 0;
			AutData.StartInterval	  	:= gA[9].AxisPeriod;
			AutData.MaxMasterVelocity	:= gr_rMachMaxSpeed_BPM ;

		(*Automat STATE 0 Basis State*)
			AutData.State[0].Event[0].Type		  := ncST_END;
			AutData.State[0].Event[0].Attribute	:= ncAT_ONCE;
      IF gA[4].Ind_bInContactZone                  AND
         (g_iMachType = C_iRS15)                   AND
         NOT(gstCycA[3].CycManTimSet.CmdSynchroOn) AND
         NOT(gstCycA[4].CycManTimSet.CmdSynchroOn) AND
         1                                         THEN
        // Start synchro with tearing and Drum in contact
        AutData.State[0].Event[0].NextState := 5;
      ELSE
        IF gA[7].bSynchroReq THEN
          AutData.State[0].Event[0].NextState := 1;
        ELSE
          AutData.State[0].Event[0].NextState := 3;
        END_IF
      END_IF

      rTemp_[0] := gA[7].PositionDeg ;
      rTemp_[1] := gA[9].PositionDeg ;

      rSlave_AxisPeriod := gA[7].AxisPeriod * gA[7].rRSynNum/gA[7].rRSynDen;

    // Master/Slave synchro calculation
      rOffsetDeg := gRecipeActive.rDrum_PhasMasterDeg ;
      // Pos Master in Slave range
      rTemp_[2] := gA[7].rRSynNum/gA[7].rRSynDen * gA[9].PositionDeg ;
      // Slave distance to be synchronized
      rTemp_[3] := rTemp_[2] - gA[7].PositionDeg + rOffsetDeg ;
      rSlCompDist := rTemp_[3] ;
      IF rSlCompDist > 180*gA[7].rRSynNum/gA[7].rRSynDen THEN
        rSlCompDist := rSlCompDist - 360*gA[7].rRSynNum/gA[7].rRSynDen ;
      END_IF ;
      IF rSlCompDist < -180*gA[7].rRSynNum/gA[7].rRSynDen THEN
        rSlCompDist := rSlCompDist + 360*gA[7].rRSynNum/gA[7].rRSynDen ;
      END_IF ;

		//Automat STATE 1 Master/Slave Absolute Phase Correction
      AutData.State[1].MasterParID     := MasterParID ;
			AutData.State[1].CamProfileIndex := 16#FFFF;
			AutData.State[1].MasterFactor		 := REAL_TO_UDINT(gA[9].AxisPeriod*2);
			AutData.State[1].SlaveFactor		 := REAL_TO_UDINT((rSlave_AxisPeriod*2)+(rSlCompDist*gA[7].UnitsPerDeg));
			AutData.State[1].CompMode			   := ncOFF;

      AutData.State[1].Event[0].Type      := ncST_END;
      AutData.State[1].Event[0].Attribute := ncST_END;
      AutData.State[1].Event[0].NextState := 3;

      AutData.State[1].Event[1].Type      := ncSIGNAL1;
      AutData.State[1].Event[1].Attribute := ncAT_ONCE;
      AutData.State[1].Event[1].NextState := 4;

		(*//Automat STATE 2 Master/Slave Transition
      AutData.State[2].MasterParID        := MasterParID ;
			AutData.State[2].CamProfileIndex	  := 16#FFFF;
			AutData.State[2].MasterFactor		    := REAL_TO_UDINT(gA[9].AxisPeriod/2);
			AutData.State[2].SlaveFactor	    	:= REAL_TO_UDINT(gA[7].AxisPeriod/2);
			AutData.State[2].CompMode			      := ncONLYCOMP;
			AutData.State[2].MasterCompDistance := gA[9].AxisPeriod-AutData.State[2].MasterFactor;
			AutData.State[2].SlaveCompDistance	:= gA[3].AxisPeriod-AutData.State[2].SlaveFactor;
			AutData.State[2].ExtendedCompLimits := ncOFF;*)

			AutData.State[2].Event[0].Type		  := ncST_END;
			AutData.State[2].Event[0].Attribute	:= ncST_END;
			AutData.State[2].Event[0].NextState	:= 3;

		//Automat STATE 3 Master/Slave Run
      AutData.State[3].MasterParID     := MasterParID ;
			AutData.State[3].CamProfileIndex := 16#FFFF;
			AutData.State[3].MasterFactor		 := REAL_TO_UDINT(gA[9].AxisPeriod);
			AutData.State[3].SlaveFactor		 := REAL_TO_UDINT(rSlave_AxisPeriod);
			AutData.State[3].CompMode			   := ncOFF;

			AutData.State[3].Event[0].Type		  := ncST_END;
			AutData.State[3].Event[0].Attribute	:= ncST_END;
			AutData.State[3].Event[0].NextState	:= 3;

      AutData.State[3].Event[1].Type      := ncSIGNAL1;
      AutData.State[3].Event[1].Attribute := ncAT_ONCE;
      AutData.State[3].Event[1].NextState := 4;

    //Automat STATE 4 Master/Slave Timing setting
      AutData.State[4].MasterParID     := uiMasterParID1 ;
      AutData.State[4].CamProfileIndex := 16#FFFF;
      AutData.State[4].MasterFactor    := REAL_TO_UDINT(gA[4].AxisPeriod);
      AutData.State[4].SlaveFactor     := REAL_TO_UDINT(gA[7].AxisPeriod);
      AutData.State[4].CompMode        := ncOFF;

      AutData.State[4].Event[0].Type      := ncST_END+ncNEGATIVE;
      AutData.State[4].Event[0].Attribute := ncST_END;
      AutData.State[4].Event[0].NextState := 4;

      AutData.State[4].Event[2].Type      := ncSIGNAL2 ;
      AutData.State[4].Event[2].Attribute := ncAT_ONCE ;
      AutData.State[4].Event[2].NextState := 3 ;

    //Automat STATE 1 Master/Slave Absolute Phase Correction in case Holding in contact with Drum
      rSPMaPos := (gA[7].PositionDeg - rOffsetDeg)/(gA[7].rRSynNum/gA[7].rRSynDen) ;
      rTemp_[6] := rSPMaPos - gA[9].PositionDeg ;
      rMaCompDist := H_FC_Modulus (
                          IN_rMod := (360 * gA[7].rRSynNum/gA[7].rRSynDen) ,
                          IN_rVar := rTemp_[6]
                                  ) ;
      iiMasterFactor5 := REAL_TO_UDINT(rMaCompDist*gA[4].UnitsPerDeg);
      IF iiMasterFactor5 < 1 THEN
        iiMasterFactor5 := REAL_TO_UDINT(gA[4].AxisPeriod) ;
        iiSlaveFactor5  := REAL_TO_UDINT(gA[7].AxisPeriod) ;
      ELSE
        iiSlaveFactor5  := 0 ;
      END_IF
      AutData.State[5].MasterParID     := MasterParID ;
      AutData.State[5].CamProfileIndex := 16#FFFF;
      AutData.State[5].MasterFactor    := iiMasterFactor5;
      AutData.State[5].SlaveFactor     := iiSlaveFactor5;
      AutData.State[5].CompMode        := ncOFF;

      AutData.State[5].Event[0].Type      := ncST_END;
      AutData.State[5].Event[0].Attribute := ncST_END;
      AutData.State[5].Event[0].NextState := 3;

      AutData.State[5].Event[1].Type      := ncSIGNAL1;
      AutData.State[5].Event[1].Attribute := ncAT_ONCE;
      AutData.State[5].Event[1].NextState := 4;

			MC_BR_AutControl_0.Enable 		 := 1;
			MC_BR_AutControl_0.AdrAutData  := ADR(AutData);
			MC_BR_AutControl_0.InitAutData := 1;
	END_IF
			(* wait for initialization done or restart *)
			IF ((MC_BR_AutControl_0.AutDataInitialized=1) AND (Synch_Request)) THEN
				MC_BR_AutControl_0.InitAutData := 0;
				MC_BR_AutControl_0.Enable :=1;
				AutomatStart := 1;
        uiMC_BR_AutControl_0_MemoErrorID := 0 ;
			END_IF
			(* check if error occured *)
			IF (MC_BR_AutControl_0.ErrorID <> 0) THEN
				MC_BR_AutControl_0.Enable := 0 ;
        uiMC_BR_AutControl_0_MemoErrorID := MC_BR_AutControl_0.ErrorID ;
			END_IF

	(******************** ENABLE CAM-AUTOMAT **********************)

	IF (AutomatStart) THEN
			MC_BR_AutControl_0.Start := 1;
			AutomatStart := 0;
	END_IF

	IF (NOT Synch_Request) THEN
			MC_BR_AutControl_0.Stop := 1;
			MC_BR_AutControl_0.Start := 0;
      ParID_Ready := 0;
      ParID_Ready1 := 0;
			IF (MC_BR_AutControl_0.Running=0) THEN
				MC_BR_AutControl_0.Enable := 0;
				MC_BR_AutControl_0.Stop := 0;
			END_IF
   //*************************************************
   // D.M. 26/01/2012 RS26 Pyrollpack_14661 added because after guard fault it happened that Stop=1 and MC_BR_AutControl_0.Enable => not possible to finish MC_BR_AutControl_0 => program locked
      IF MC_BR_AutControl_0.Stop        AND
         NOT(MC_BR_AutControl_0.Enable) THEN
        MC_BR_AutControl_0.Enable := 1 ;
      END_IF
   //*************************************************
	END_IF

	gA[7].Ind_AutomatEnabled:=MC_BR_AutControl_0.Enable;
	gA[7].Ind_CurrentAutomatState:=MC_BR_AutControl_0.ActualStateIndex;
  gA[7].Ind_bSynchroOK := (MC_BR_AutControl_0.ActualStateIndex >= 3) AND gA[7].Ind_SynchronizedMotion ; ;

	(********************** MC_AUTCONTROL *************************)
	MC_BR_AutControl_0.Slave:= gA[7].Ident;
	MC_BR_AutControl_0();

END_PROGRAM
```

### Program Logical/BagMachine_Section/Drum/Axis7/A7_Ref (IEC) - Reference Routine

#### A7_Ref.var
```iecst
(********************************************************************
 * COPYRIGHT -- Microsoft
 ********************************************************************
 * Program: A7_Ref
 * File: A7_Ref.var
 * Author: pkiel
 * Created: July 19, 2011
 ********************************************************************
 * Local variables of program A7_Ref
 ********************************************************************)
VAR
	HGW_2StepMove_0 : HGW_2StepMove;
	MC_Home_0 : MC_Home;
	MC_Home_1 : MC_Home;
	MC_MoveAdditive_0 : MC_MoveAdditive;
	Ref_Seq : ARRAY[0..10] OF BOOL;
  bTest : BOOL ;
END_VAR
```

#### A7_RefCyclic.ld
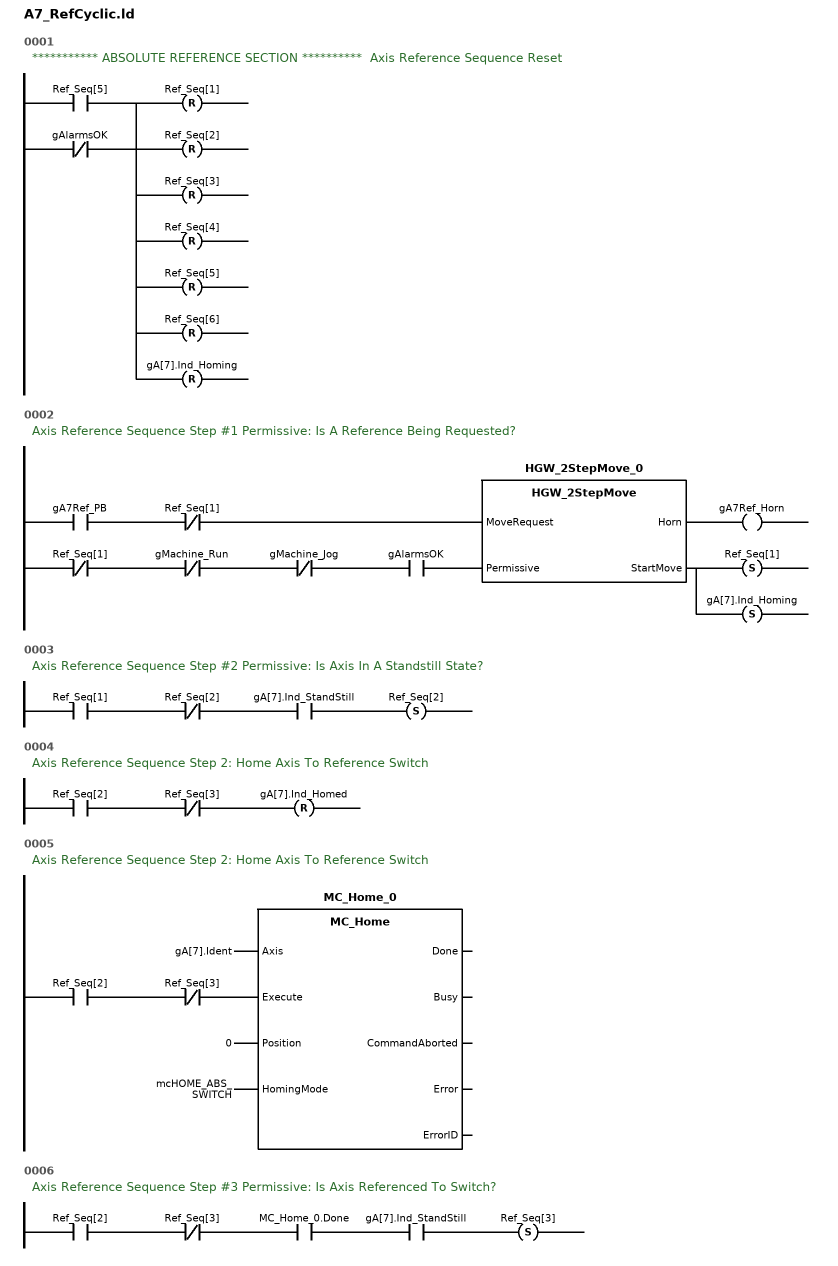
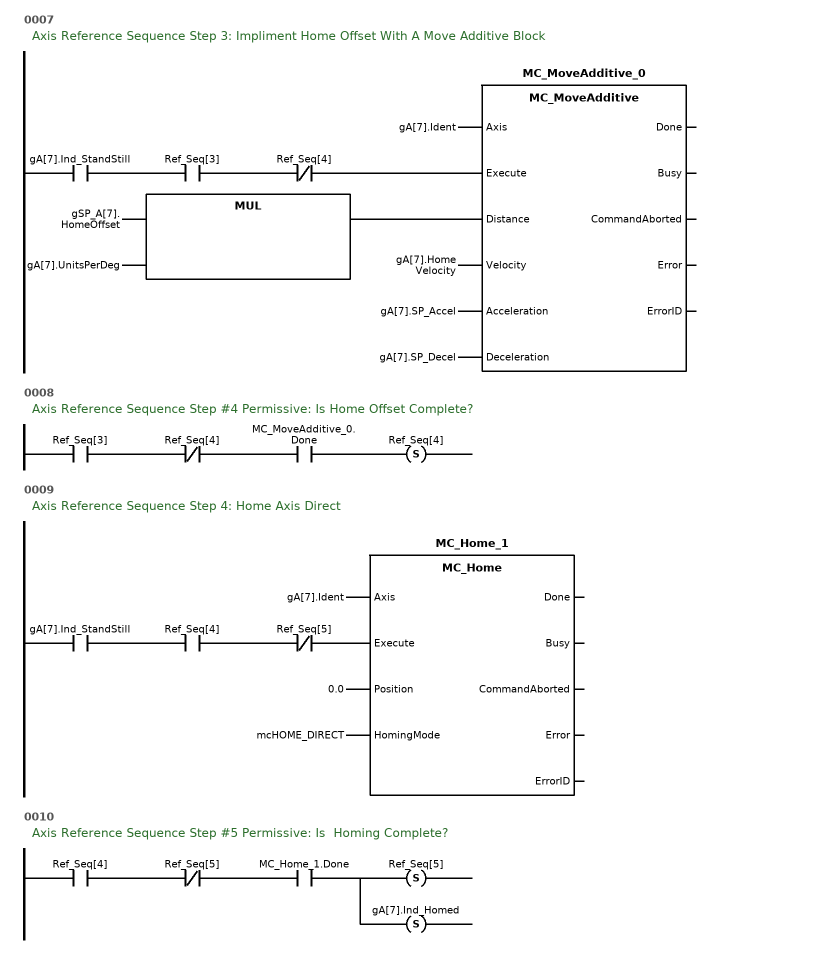
Ladder, written as Structured Text:
```iecst
(********************************************************************
 * COPYRIGHT -- Microsoft
 ********************************************************************
 * Program: A7_Ref
 * File: A7_RefCyclic.ld
 * Author: pkiel
 * Created: July 19, 2011
 ********************************************************************
 * Implementation of program A7_Ref
 ********************************************************************)

PROGRAM _CYCLIC
VAR
    _p1 : BOOL;
    _p2 : BOOL;
END_VAR
(* Network 1: *********** ABSOLUTE REFERENCE SECTION **********  Axis Reference Sequence Reset *)
_p1 := Ref_Seq[5];
IF Ref_Seq[5] OR NOT gAlarmsOK THEN Ref_Seq[1] := FALSE; END_IF;
IF _p1 OR NOT gAlarmsOK THEN
    Ref_Seq[2] := FALSE;
    Ref_Seq[3] := FALSE;
    Ref_Seq[4] := FALSE;
    Ref_Seq[5] := FALSE;
    Ref_Seq[6] := FALSE;
    gA[7].Ind_Homing := FALSE;
END_IF;

(* Network 2: Axis Reference Sequence Step #1 Permissive: Is A Reference Being Requested? *)
HGW_2StepMove_0(MoveRequest := gA7Ref_PB AND NOT Ref_Seq[1], Permissive := NOT Ref_Seq[1] AND NOT gMachine_Run AND NOT gMachine_Jog AND gAlarmsOK);
gA7Ref_Horn := HGW_2StepMove_0.Horn;
IF HGW_2StepMove_0.StartMove THEN
    Ref_Seq[1] := TRUE;
    gA[7].Ind_Homing := TRUE;
END_IF;

(* Network 3: Axis Reference Sequence Step #2 Permissive: Is Axis In A Standstill State? *)
IF Ref_Seq[1] AND NOT Ref_Seq[2] AND gA[7].Ind_StandStill THEN Ref_Seq[2] := TRUE; END_IF;

(* Network 4: Axis Reference Sequence Step 2: Home Axis To Reference Switch *)
IF Ref_Seq[2] AND NOT Ref_Seq[3] THEN gA[7].Ind_Homed := FALSE; END_IF;

(* Network 5: Axis Reference Sequence Step 2: Home Axis To Reference Switch *)
MC_Home_0(Axis := gA[7].Ident, Execute := Ref_Seq[2] AND NOT Ref_Seq[3], Position := 0, HomingMode := mcHOME_ABS_SWITCH);

(* Network 6: Axis Reference Sequence Step #3 Permissive: Is Axis Referenced To Switch? *)
IF Ref_Seq[2] AND NOT Ref_Seq[3] AND MC_Home_0.Done AND gA[7].Ind_StandStill THEN
    Ref_Seq[3] := TRUE;
END_IF;

(* Network 7: Axis Reference Sequence Step 3: Impliment Home Offset With A Move Additive Block *)
MC_MoveAdditive_0(Axis := gA[7].Ident, Execute := gA[7].Ind_StandStill AND Ref_Seq[3] AND NOT Ref_Seq[4], Distance := gSP_A[7].HomeOffset * gA[7].UnitsPerDeg, Velocity := gA[7].HomeVelocity, Acceleration := gA[7].SP_Accel, Deceleration := gA[7].SP_Decel);

(* Network 8: Axis Reference Sequence Step #4 Permissive: Is Home Offset Complete? *)
IF Ref_Seq[3] AND NOT Ref_Seq[4] AND MC_MoveAdditive_0.Done THEN Ref_Seq[4] := TRUE; END_IF;

(* Network 9: Axis Reference Sequence Step 4: Home Axis Direct *)
MC_Home_1(Axis := gA[7].Ident, Execute := gA[7].Ind_StandStill AND Ref_Seq[4] AND NOT Ref_Seq[5], Position := 0.0, HomingMode := mcHOME_DIRECT);

(* Network 10: Axis Reference Sequence Step #5 Permissive: Is  Homing Complete? *)
_p2 := Ref_Seq[4] AND NOT Ref_Seq[5] AND MC_Home_1.Done;
IF Ref_Seq[4] AND NOT Ref_Seq[5] AND MC_Home_1.Done THEN Ref_Seq[5] := TRUE; END_IF;
IF _p2 THEN gA[7].Ind_Homed := TRUE; END_IF;
END_PROGRAM
```

### Program Logical/BagMachine_Section/Drum/Axis7/A7_Cycle (IEC) - A new program

#### A7_CycleCyclic.st
```iecst
(********************************************************************
 * COPYRIGHT -- .
 ********************************************************************
 * Program: A7_Cycle
 * File: A7_CycleCyclic.st
 * Author: dominique
 * Created: August 01, 2011
 ********************************************************************
 * Implementation of program A7_Cycle
 ********************************************************************)

PROGRAM _CYCLIC

// Manu axis movement for timing setting

    //---------------------------------------------------------------------------------------------------------------------
    // Drum timing setting cycle
    //---------------------------------------------------------------------------------------------------------------------
    // Start cycle
    gstCycA[7].CycManTimSet.CmdStart := ( gA[7].Cmd_ManuTimSetPlus        OR
                                          gA[7].Cmd_ManuTimSetMinus )     AND
                                        ( NOT(g_bCycManTimeSetOn)         OR
                                          gstCycA[7].CycManTimSet.bSCyc ) AND
                                        gA[7].Ind_Ready                   ;
    IF gstCycA[7].CycManTimSet.CmdStart THEN
      gstCycA[7].CycManTimSet.bSCyc := 1 ;
    END_IF ;

    //----------------------------------------------------------------------
    // Cycle at rest
    IF NOT(gstCycA[7].CycManTimSet.bSCyc) AND
       1                                 THEN
      IF NOT( gstCycA[7].CycManTimSet.bFCyc ) THEN
        // Init after cycle unpropaly ended
        gstCycA[7].CycManTimSet.bFCyc := 1 ;
        gstCycA[7].CycManTimSet.bCyc  := 0 ;

        gstCycA[7].CycManTimSet.CmdMov       := 0 ;
        gstCycA[7].CycManTimSet.CmdStop      := 0 ;
        gstCycA[7].CycManTimSet.CmdSynchroOn := 0 ;
      END_IF
      gstCycA[7].CycManTimSet.iStep := 0 ;
      RETURN ;
    ELSE
    //----------------------------------------------------------------------
    // Cycle running

      // Permanent conditions
      IF NOT(gA[7].Ind_Ready)                  OR
         NOT(gstCycA[7].CycManTimSet.CmdStart) AND
         (gstCycA[7].CycManTimSet.iStep <= 2)  THEN
        gstCycA[7].CycManTimSet.bSCyc := 0 ;
        RETURN ;
      END_IF

      // Permanent actions
      stTON_01 (
            IN := ( gstCycA[7].CycManTimSet.iStep = C_iSTEP_0 ) ,
            PT := T#30ms
               ) ;
    END_IF
    //----------------------------------------------------------------------
    // Cycle steps

        CASE gstCycA[7].CycManTimSet.iStep OF

        C_iSTEP_0 :
         //----------------------------------------------
         // Etape 1 : Initialisation
         //----------------------------------------------
          IF stTON_01.Q THEN
            gstCycA[7].CycManTimSet.iStep := C_iSTEP_1 ;

            // Action Step 1
            gstCycA[7].CycManTimSet.bFCyc := 0 ;
            gstCycA[7].CycManTimSet.bCyc  := 1 ;
          END_IF

        C_iSTEP_1 :
         //----------------------------------------------
         // Etape 2 : Synchro Drum
         //----------------------------------------------
          IF TRUE THEN
            gstCycA[7].CycManTimSet.iStep := C_iSTEP_2 ;

            // Action Step 2
            gstCycA[7].CycManTimSet.CmdSynchroOn := 1 ;
          END_IF

        C_iSTEP_2 :
         //----------------------------------------------
         // Step 3 : Activation motion and Stop waiting
         //----------------------------------------------
          IF gstCycA[7].CycManTimSet.bSynchroOkSlavA[7] THEN
            gstCycA[7].CycManTimSet.iStep := C_iSTEP_3 ;

            // Action Step 3
            gstCycA[7].CycManTimSet.CmdMov  := 1 ;
            gstCycA[7].CycManTimSet.CmdStop := 0 ;
            // Stop waiting
          END_IF

        C_iSTEP_3 :
         //----------------------------------------------
         // Step 4 : Stop motion and End stop waiting
         //----------------------------------------------
          IF NOT(gstCycA[7].CycManTimSet.CmdStart) THEN
            gstCycA[7].CycManTimSet.iStep := C_iSTEP_4 ;

            // Action Step 4
            gstCycA[7].CycManTimSet.CmdMov  := 0 ;
            gstCycA[7].CycManTimSet.CmdStop := 1 ;
            // End stop waiting
          END_IF

        C_iSTEP_4 :
         //----------------------------------------------
         // Step 3 : Activation motion and Stop waiting
         // Step 5 : Cut synchro
         //----------------------------------------------
          // Condition Step3
          IF gstCycA[7].CycManTimSet.CmdStart THEN
            gstCycA[7].CycManTimSet.iStep := C_iSTEP_3 ;

            // Action Step 3
            gstCycA[7].CycManTimSet.CmdMov  := 1 ;
            gstCycA[7].CycManTimSet.CmdStop := 0 ;
            // Stop waiting
            RETURN ;
          END_IF ;
          // Condition Step5
          IF NOT(gstCycA[7].CycManTimSet.CmdStop) THEN
            gstCycA[7].CycManTimSet.iStep := C_iSTEP_5 ;

            // Action Step 5
            gstCycA[7].CycManTimSet.CmdSynchroOn := 0 ;
          END_IF

        C_iSTEP_5 :
         //----------------------------------------------
         // Step 6 : New offset calculation
         //----------------------------------------------
          IF TRUE THEN
            gstCycA[7].CycManTimSet.iStep := C_iSTEP_6 ;

            // Action Step 6
            // Memo Actual phase Offset
            rTempActPhasDeg[7]    := gRecipeActive.rDrum_PhasMasterDeg ;
            rTempActOffsetInch[7] := gRecipeActive.Drum_Offset ;
            // Update phase
            gRecipeActive.rDrum_PhasMasterDeg := gA[7].rActPhasDeg ;
            // Update Offset
            rTemp_[7] := rTempActOffsetInch[7] + (gRecipeActive.rDrum_PhasMasterDeg - rTempActPhasDeg[7])/(gA[7].rRSynNum/gA[7].rRSynDen)*gA[7].InchPerDeg ;
            gRecipeActive.Drum_Offset := H_FC_Modulus (IN_rMod := gRecipeActive.Repeat, IN_rVar := rTemp_[7]) ;
          END_IF

        C_iSTEP_6 :
         //----------------------------------------------
         // Step 0 : First step
         //----------------------------------------------
          IF TRUE THEN
            gstCycA[7].CycManTimSet.iStep := C_iSTEP_0 ;

            // Action Step 0
            gstCycA[7].CycManTimSet.bSCyc := 0 ;
            gstCycA[7].CycManTimSet.bFCyc := 1 ;
            gstCycA[7].CycManTimSet.bCyc  := 0 ;
          END_IF
        END_CASE
    //---------------------------------------------------------------------------------------------------------------------

END_PROGRAM
```

#### A7_CycleInit.st
```iecst
(********************************************************************
 * COPYRIGHT -- .
 ********************************************************************
 * Program: A7_Cycle
 * File: A7_CycleInit.st
 * Author: dominique
 * Created: August 01, 2011
 ********************************************************************
 * Implementation of program A7_Cycle
 ********************************************************************)

PROGRAM _INIT

  gstCycA[7].CycManTimSet.uiMasterParID := 428 ; // ParID 428 = CTRL Position controller: Input set position (in case real axis)

END_PROGRAM
```

### Program Logical/BagMachine_Section/EntryPull/Axis5/A5_Basic

#### A5_BasicInit.st
```iecst
(********************************************************************
 * COPYRIGHT -- Microsoft
 ********************************************************************
 * Program: A5_Basic
 * File: A5_BasicInit.st
 * Author: pkiel
 * Created: July 13, 2011
 ********************************************************************
 * Implementation of program A5_Basic
 ********************************************************************)

PROGRAM _INIT

	(* Axis Setpoint Variables *)
		gA[5].SP_MotorPPR := 14400;
		gA[5].SP_GearBoxInput:= 5;
		gA[5].SP_GearBoxOutput:= 2;
		gA[5].AxisPeriod := (gA[5].SP_MotorPPR*gA[5].SP_GearBoxInput/gA[5].SP_GearBoxOutput);
		gA[5].UnitsPerDeg := gA[5].AxisPeriod/360;
		gA[5].SP_Accel := 0.2*gA[5].AxisPeriod;
		gA[5].SP_Decel := 0.4*gA[5].AxisPeriod;
		gA[5].SP_EStopDecel := 1000.0*gA[5].AxisPeriod; // Stop axis from 1000 tr/min in 1s
		(* Theoretical Perimeter = 400mm *)
		gA[5].UnitsPerInch := gA[5].AxisPeriod*25.4/g_rSizeEntryPullRol_mm ;
    gA[5].rSP_CorPosVel := 0.0 ;
    gA[5].rSP_OverrideV := 1.0 ;
    gA[5].rSP_OverrideA := 1.0 ;
    gA[5].Cmd_EStopDisable := 0 ;

	(* access master axis *)
		AxisErrorNcAccess := ncaccess(ncACP10MAN, ADR('Axis5'), ADR(gA[5].Ident));

	(* Trigger Initialization Of ModPosition *)
		InitModPosition:=1;
END_PROGRAM
```

### Program Logical/BagMachine_Section/EntryPull/Axis5/A5_Draw

#### A5_DrawCyclic.st
```iecst
(********************************************************************
 * COPYRIGHT -- Microsoft
 ********************************************************************
 * Program: A5_Draw
 * File: A5_DrawCyclic.st
 * Author: pkiel
 * Created: July 13, 2011
 ********************************************************************
 * Implementation of program A5_Draw
 ********************************************************************)

PROGRAM _CYCLIC

(* Draw Setpoint Limits *)
	gRecipeActive.Entry_Draw := LIMIT(-100,gRecipeActive.Entry_Draw,100);

  // Lock Entry Web Draw in case Reg Enable
  IF EDGENEG(gReg[5].Enable) THEN
    HMI_rEntry_Draw_Set := gRecipeActive.Entry_Draw ;
  END_IF
  IF gReg[5].Enable THEN
    iLockEntryWebDraw := 2 ; // Lock
    iBackColor := gGray1 + gBlack * 256 ;
    HMI_rEntry_Draw_Set := 0.0 ;
    rEntry_Draw_SP := 0.0 ;
  ELSE
    iLockEntryWebDraw := 0 ; // Free
    iBackColor := gWhite + gBlack * 256 ;
    gRecipeActive.Entry_Draw := HMI_rEntry_Draw_Set ;
    rEntry_Draw_SP := gRecipeActive.Entry_Draw ;
  END_IF

(* Manual Draw Calculations *)
  IF (((rEntry_Draw_SP <> Draw_Old) OR (NOT First) OR gRepeatChange) AND gA[5].Ind_SynchronizedMotion) THEN
    gA5_GearValue := gA[5].UnitsPerInch * gRecipeActive.Repeat * (1+(gr_rMaxRangeWebDraw * 0.01 * rEntry_Draw_SP * 0.01));
    Draw_Old := rEntry_Draw_SP ;
    First :=1;
    IF(gA[5].Ind_SynchronizedMotion) THEN
      gA[5].Cmd_SynchronizedMotionUpdate := NOT(gReg[5].Enable) ;
    END_IF
  END_IF

END_PROGRAM
```

#### A5_DrawInit.st
```iecst
(********************************************************************
 * COPYRIGHT -- .
 ********************************************************************
 * Program: A5_Draw
 * File: A5_DrawInit.st
 * Author: dominique
 * Created: January 06, 2012
 ********************************************************************
 * Implementation of program NewProgram
 ********************************************************************)

PROGRAM _INIT

    HMI_rEntry_Draw_Set := gRecipeActive.Entry_Draw ;

END_PROGRAM
```

### Data object Logical/BagMachine_Section/EntryPull/Axis5/A5_Init (Ax)

#### A5_Init.ax
```
InitParameter (Version=2.24.0, NcSwId=ACP10)
  ACP10AXIS_typ:
    dig_in:
      level:
        reference = ncACTIV_HI
        pos_hw_end = ncACTIV_HI
        neg_hw_end = ncACTIV_HI
        trigger1 = ncACTIV_HI
        trigger2 = ncACTIV_HI
    encoder_if:
      parameter:
        count_dir = ncSTANDARD
        scaling:
          load:
            units = 14400  // Units at the load = 36000 x 2 / 5 
            rev_motor = 1  // Motor revolutions = 1
    limit:
      parameter:
        v_pos = 720000.0
        v_neg = 720000.0
        a1_pos = 5e+006
        a2_pos = 5e+006
        a1_neg = 5e+006
        a2_neg = 5e+006
        t_jolt = 0.0
        t_in_pos = 0.0
        pos_sw_end = 8388607
        neg_sw_end = -8388608
        ds_warning = 500.0
        ds_stop = 1000.0
        a_stop = 1e+030
        dv_stop = 0
        dv_stop_mode = ncOFF
    controller:
      mode = ncPOSITION
      position:
        kv = 350.0
        tn = 0.0
        t_predict = 0.0004
        t_total = 0.0004
        p_max = 1e+030
        i_max = 0.0
      speed:
        kv = 30.0
        tn = 0.0
        t_filter = 0.0
        isq_filter1:
          type = ncOFF
          a0 = 0.0
          a1 = 0.0
          b0 = 0.0
          b1 = 0.0
          b2 = 0.0
          c0_par_id = 0
          c1_par_id = 0
        isq_filter2:
          type = ncOFF
          a0 = 0.0
          a1 = 0.0
          b0 = 0.0
          b1 = 0.0
          b2 = 0.0
          c0_par_id = 0
          c1_par_id = 0
        isq_filter3:
          type = ncOFF
          a0 = 0.0
          a1 = 0.0
          b0 = 0.0
          b1 = 0.0
          b2 = 0.0
          c0_par_id = 0
          c1_par_id = 0
      uf:
        type = ncLINEAR
        auto_config = ncMOTOR_PAR
        u0 = 0.0
        un = 0.0
        fn = 50.0
        k_f_slip = 0.0
      ff:
        torque_load = 0.0
        torque_pos = 0.0
        torque_neg = 0.0
        kv_torque = 0.0
        inertia = 0.0
        t_filter_a = 0.0
    move:
      stop:
        parameter[0]:
          decel_ramp = ncA_LIMIT
          controller = ncON
        parameter[1]:
          decel_ramp = ncA_LIMIT
          controller = ncON
        parameter[2]:
          decel_ramp = ncA_LIMIT
          controller = ncON
        parameter[3]:
          decel_ramp = ncA_LIMIT
          controller = ncON
        quickstop:
          decel_ramp = ncA_LIMIT
        drive_error:
          decel_ramp = ncA_LIMIT
      homing:
        parameter:
          s = 0
          v_switch = 5000.0
          v_trigger = 500.0
          a = 50000.0
          mode = ncHOME_OFFSET
          edge_sw = ncPOSITIVE
          start_dir = ncPOSITIVE
          trigg_dir = ncPOSITIVE
          ref_pulse = ncOFF
          tr_s_block = 0.0
      basis:
        parameter:
          v_pos = 36000.0
          v_neg = 100000.0
          a1_pos = 50000.0
          a2_pos = 50000.0
          a1_neg = 50000.0
          a2_neg = 50000.0
    message:
      text:
        parameter:
          format = ncBREAK
          columns = 80
          data_modul = Error_Eng
```

### A5_Par.apt
```
AcoposParameterTable:
  Root Parameters:
    110 = ncSW_OFF (Name=CMD_SIMULATION)  // Simulation mode: Command
    128 = 1 (Name=SGEN_SW_END_IGNORE)  // SGEN_SW_END_IGNORE
    390 = 565 (Name=UDC_NOMINAL, Unit=V)  // CTRL DC bus: Nominal voltage
```

### Program Logical/BagMachine_Section/EntryPull/EntryNip

#### EntryNipCyclic.ld
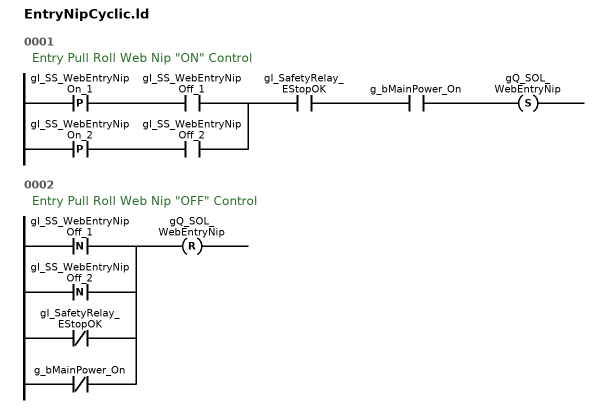
Ladder, written as Structured Text:
```iecst
(********************************************************************
 * COPYRIGHT -- Microsoft
 ********************************************************************
 * Program: EntryNip
 * File: EntryNipCyclic.ld
 * Author: pkiel
 * Created: July 20, 2011
 ********************************************************************
 * Implementation of program EntryNip
 ********************************************************************)

PROGRAM _CYCLIC
VAR
    _e1 : R_TRIG;
    _e2 : R_TRIG;
    _e3 : F_TRIG;
    _e4 : F_TRIG;
END_VAR
(* Network 1: Entry Pull Roll Web Nip "ON" Control *)
_e1(CLK := gI_SS_WebEntryNipOn_1);
_e2(CLK := gI_SS_WebEntryNipOn_2);
IF ((_e1.Q AND gI_SS_WebEntryNipOff_1) OR (_e2.Q AND gI_SS_WebEntryNipOff_2)) AND gI_SafetyRelay_EStopOK AND g_bMainPower_On THEN
    gQ_SOL_WebEntryNip := TRUE;
END_IF;

(* Network 2: Entry Pull Roll Web Nip "OFF" Control *)
_e3(CLK := gI_SS_WebEntryNipOff_1);
_e4(CLK := gI_SS_WebEntryNipOff_2);
IF _e3.Q OR _e4.Q OR NOT gI_SafetyRelay_EStopOK OR NOT g_bMainPower_On THEN
    gQ_SOL_WebEntryNip := FALSE;
END_IF;
END_PROGRAM
```

### Program Logical/BagMachine_Section/EntryPull/Registration/A5_Reg1 (IEC)

#### A5_Reg1Cyclic.st - Cyclic code
```iecst
(********************************************************************
 * COPYRIGHT -- Microsoft
 ********************************************************************
 * Program: A5_Reg1
 * File: A5_Reg1Cyclic.st
 * Author: pkiel
 * Created: July 19, 2011
 ********************************************************************
 * Implementation of program A5_Reg1
 ********************************************************************)

PROGRAM _CYCLIC

(*** REGISTRATION PROGRAM FOR MARK TO MACHINE REGISTRATION USED ON A DRAWROLL ***)
(*** Note: Since both the exit pull roll is slaved to the entry pull roll, the registration correction
	only needs to be sent into the entry pull roll axis.  ***)

(************************ REGISTRATION CAPTURE SECTION **********************)

(* Registration TouchProbe Capture 0...Used To Capture Master For Calculating Registration Correction *)
	MC_BR_TouchProbe_0.Axis:=gA[9].Ident;
	MC_BR_TouchProbe_0.TriggerInput:=TriggerRef_0;
	MC_BR_TouchProbe_0.Enable:=gReg[5].Enable;
	MC_BR_TouchProbe_0.Period:=gRecipeActive.Repeat*gA[9].UnitsPerInch*gReg[5].SP_Format;
	MC_BR_TouchProbe_0.WindowNegative:=gRecipeActive.Repeat*gA[9].UnitsPerInch*0.5*gReg[5].SP_Format;
	MC_BR_TouchProbe_0.WindowPositive:=MC_BR_TouchProbe_0.WindowNegative;
	MC_BR_TouchProbe_0.Mode:=68;
	MC_BR_TouchProbe_0();
rRecordedPeriodicValue[0] := MC_BR_TouchProbe_0.RecordedPeriodicValue;

(* Registration TouchProbe Capture 1...Used To Capture Slave For Qualifying Registration Marks & Calculating Length *)
	MC_BR_TouchProbe_1.Axis:=gA[5].Ident;
	MC_BR_TouchProbe_1.TriggerInput:=TriggerRef_1;
	MC_BR_TouchProbe_1.Enable:=gReg[5].Enable;
	MC_BR_TouchProbe_1.Period:=gRecipeActive.Repeat*gA[5].UnitsPerInch*gReg[5].SP_Format;
	MC_BR_TouchProbe_1.PeriodChange:=(gReg[5].LengthAverage*gA[5].UnitsPerInch*gReg[5].SP_Format)-MC_BR_TouchProbe_1.Period;
	MC_BR_TouchProbe_1.WindowNegative:=gReg[5].SP_Tolerance*gA[5].UnitsPerInch;
	MC_BR_TouchProbe_1.WindowPositive:=MC_BR_TouchProbe_1.WindowNegative;
	MC_BR_TouchProbe_1.Mode:=mcSHIFT_FROM_RESULT+mcUSE_FIRST_TRIGGER_POS;
	MC_BR_TouchProbe_1();

(* Detect First Mark *)
	IF ((MC_BR_TouchProbe_1.ProbeCounter = 1)AND(NOT gReg[5].MarkFirst)) THEN
		gReg[5].MarkFirst:=1;
		FirstCapture:=MC_BR_TouchProbe_0.RecordedPeriodicValue;
	END_IF;

(* Detect Probe Counter 0 Change *)
	IF (MC_BR_TouchProbe_0.ProbeCounter <> ProbeCounter0_Old) THEN
		ProbeCounter0_Change:=1;
		ProbeCounter0_Old:=MC_BR_TouchProbe_1.ProbeCounter;
	END_IF

(* Detect Probe Counter 1 Change *)
	IF (MC_BR_TouchProbe_1.ProbeCounter <> ProbeCounter1_Old) THEN
		ProbeCounter1_Change:=1;
		ProbeCounter1_Old:=MC_BR_TouchProbe_1.ProbeCounter;
	END_IF

(* Detect Change In Both Probe Counters *)
	IF (ProbeCounter0_Change AND ProbeCounter1_Change) THEN
		ProbeCounter_Change:=1;
		ProbeCounter0_Change:=0;
		ProbeCounter1_Change:=0;
	ELSE
		ProbeCounter_Change:=0;
	END_IF;

(* Detect Good Mark *)
	IF (gReg[5].MarkFirst AND ProbeCounter_Change AND gReg[5].Enable) THEN
		gReg[5].MarkGood:=1;
		gReg[5].MarkGoodNew:=1;
		gReg[5].MarkMissed:=0;
		gReg[5].Ind_General:=2;
		gReg[5].MarkGoodCount:=gReg[5].MarkGoodCount+1;
		gReg[5].LengthActual:=gRecipeActive.Repeat-((MC_BR_TouchProbe_1.DeltaExpectedValue/gA[5].UnitsPerInch)/gReg[5].SP_Format);
	ELSE
		gReg[5].MarkGood:=0;
	END_IF;

(* Detect Missed Trigger Change *)
	IF (MC_BR_TouchProbe_1.MissedTriggers <> MissedTriggers_Old) THEN
		MissedTrigger_Change:=1;
		MissedTriggers_Old:=MC_BR_TouchProbe_1.MissedTriggers;
	ELSE
		MissedTrigger_Change:=0;
	END_IF;

	(* Detect Missed Mark *)
	IF (MissedTrigger_Change AND gReg[5].Enable) THEN
		gReg[5].MarkMissed:=1;
		gReg[5].MarkMissedNew:=1;
		gReg[5].MarkMissedCount:=gReg[5].MarkMissedCount+1;
		gReg[5].Ind_General:=1;
	END_IF;

(**** REGISTRATION CORRECTION CALCULATION SECTION ****)

(* Calculate Expected Capture Value *)
	Period:=gRecipeActive.Repeat*gA[9].UnitsPerInch;
	ExpectedCapture:=FirstCapture-(gReg[5].SP_Offset*gA[9].UnitsPerInch);
	IF (ExpectedCapture>Period) THEN
		ExpectedCapture:=ExpectedCapture-Period;
	END_IF;
	IF (ExpectedCapture<0) THEN
		ExpectedCapture:=ExpectedCapture+Period;
	END_IF;

rRecordedPeriodicValue[1] := MC_BR_TouchProbe_0.RecordedPeriodicValue;

(* Calculate Correction *)
	HGW_RegCorrectABS_0.Enable:=gReg[5].Enable;
	HGW_RegCorrectABS_0.NewCapture:=MC_BR_TouchProbe_0.RecordedPeriodicValue;
	HGW_RegCorrectABS_0.Expected:=ExpectedCapture;
	HGW_RegCorrectABS_0.Period:=Period;
	HGW_RegCorrectABS_0.WeightingFactor:=gReg[5].SP_WeightingFactor;
	HGW_RegCorrectABS_0.MaxCorrection:=gReg[5].SP_MaximumCorrection*gA[9].UnitsPerInch*gReg[5].SP_Format;
	HGW_RegCorrectABS_0.Execute:=gReg[5].MarkGood;
	HGW_RegCorrectABS_0();

	IF (gReg[5].MarkGood) THEN
		gReg[5].LengthCorrection:=HGW_RegCorrectABS_0.Correction/gA[9].UnitsPerInch;
		gReg[5].CorrectionMax:=HGW_RegCorrectABS_0.MaxCorrectionExceeded;
	END_IF;

(************************ REGISTRATION CORRECTION/PHASE **********************)

(* Only Enable Phasing When In Synch Mode *)
	IF (gA[5].Ind_SynchronizedMotion) THEN
    MC_BR_Phasing_1.Enable:=1 AND NOT(bTest) ;
	ELSE;
		MC_BR_Phasing_1.Enable:=0;
	END_IF;
	MC_BR_Phasing_1.Shift:=HGW_RegCorrectABS_0.Correction;
	MC_BR_Phasing_1.Velocity:=1000000;
	MC_BR_Phasing_1.Acceleration:=1000000;
	MC_BR_Phasing_1.ApplicationDistance:= 0.75*gRecipeActive.Repeat*gA[9].UnitsPerInch*gReg[5].SP_Format;
	MC_BR_Phasing_1.Slave:=gA[5].Ident;
	MC_BR_Phasing_1.ApplicationMode:=mcMASTER_DISTANCE_BASED;
	MC_BR_Phasing_1.ShiftMode:=mcRELATIVE;
	MC_BR_Phasing_1.InitData:=gReg[5].MarkGood;
	MC_BR_Phasing_1();

END_PROGRAM
```

#### A5_Reg1.var - Local variables
```iecst
(********************************************************************
 * COPYRIGHT -- Microsoft
 ********************************************************************
 * Program: A5_Reg1
 * File: A5_Reg1.var
 * Author: pkiel
 * Created: July 19, 2011
 ********************************************************************
 * Local variables of program A5_Reg1
 ********************************************************************)
VAR
	ExpectedCapture : REAL;
	FirstCapture : REAL;
	HGW_RegCorrectABS_0 : HGW_RegCorrectABS;
	MC_BR_Phasing_1 : MC_BR_Phasing;
	MC_BR_TouchProbe_0 : MC_BR_TouchProbe;
	MC_BR_TouchProbe_1 : MC_BR_TouchProbe;
	MissedTrigger_Change : BOOL;
	MissedTriggers_Old : UDINT;
	Period : REAL;
	ProbeCounter_Change : BOOL;
	ProbeCounter0_Change : BOOL;
	ProbeCounter0_Old : UDINT;
	ProbeCounter1_Change : BOOL;
	ProbeCounter1_Old : UDINT;
	TriggerRef_0 : MC_BR_TRIGGER_REF;
	TriggerRef_1 : MC_BR_TRIGGER_REF;

  bTest : BOOL ;
  iCptFormat : INT ;
  rRecordedPeriodicValue : ARRAY[0..9] OF REAL ;
END_VAR
```

### Program Logical/BagMachine_Section/EntryPull/Registration/A5_Reg2 (IEC)

#### A5_Reg2Cyclic.st - Cyclic code
```iecst
(********************************************************************
 * COPYRIGHT -- Microsoft
 ********************************************************************
 * Program: A5_Reg2
 * File: A5_Reg2Cyclic.st
 * Author: pkiel
 * Created: July 19, 2011
 ********************************************************************
 * Implementation of program A5_Reg2
 ********************************************************************)

PROGRAM _CYCLIC

(**** DRAWROLL GENERAL REGISTRATION STATUS & CONTROL SECTION ****)

(*** Registration Limits ***)
	gReg[5].SP_Tolerance:=LIMIT(0.375,gReg[5].SP_Tolerance,(0.5*gRecipeActive.Repeat));
	gReg[5].SP_Offset:=LIMIT(-gRecipeActive.Repeat,gReg[5].SP_Offset,gRecipeActive.Repeat);
	gReg[5].SP_Format:=LIMIT(1,gReg[5].SP_Format,4);
	gReg[5].SP_WeightingFactor:=LIMIT(0.3,gReg[5].SP_WeightingFactor,1);

(* Turn Off Registration On A Web Break *)
	IF (EDGENEG(gBagMachine_WebBreakOK)) THEN
		gReg[5].Enable := 0;
	END_IF

(*Registration OFF *)
	IF (NOT gReg[5].Enable) THEN
		gReg[5].MarkFirst:=0;
		gReg[5].MarkMissed:=0;
		gReg[5].Ind_General:=0;
		FirstAverage:=0;
		gReg[5].LengthAverage:=gRecipeActive.Repeat;
	END_IF

(* Registration Initialization *)
	IF(gReg[5].Enable AND (NOT gReg[5].MarkFirst)) THEN
		gReg[5].Ind_General:=1;
		gReg[5].LengthCorrection:=0;
		gReg[5].LengthActual:=gRecipeActive.Repeat;
		gReg[5].SP_Offset:=0;
	END_IF

(*Reset Counts When Registration Is Turned On *)
	IF (EDGEPOS(gReg[5].Enable)) THEN
		gReg[5].MarkMissedCount:=0;
		gReg[5].MarkGoodCount:=0;
	END_IF

	(* Registration HMI Button Display *)
	CASE gReg[5].Ind_General OF
		0:
			gReg[5].Ind_Text:=0;
			Background:=gBlue;
			Foreground:=gWhite;
		1:
			gReg[5].Ind_Text:=1;
			Background:=gYellow;
			Foreground:=gBlack;
		2:
			gReg[5].Ind_Text:=2;
			Background:=gGreen;
			Foreground:=gBlack;
	ELSE
		gReg[5].Ind_General:=0;
	END_CASE;
	gReg[5].Ind_Color:=Background+Foreground*256;

(**** REGISTRATION AVERAGING SECTION ****)

(* Registration Averaging Calculations *)
	IF (gReg[5].MarkGoodNew AND FirstAverage) THEN
		HGW_Average_0.ActualLength:=gReg[5].LengthActual;
		HGW_Average_0.Execute:=1;
	ELSE
		HGW_Average_0.Execute:=0;
	END_IF;
	IF (gReg[5].MarkGoodNew) THEN
		FirstAverage:=1;
	END_IF;

(* Registration Averaging Function Block *)
	HGW_Average_0.Enable:=gReg[5].Enable;
	HGW_Average_0.ProgramLength:=gRecipeActive.Repeat;
	HGW_Average_0();
	IF (gReg[5].Enable) THEN
		gReg[5].LengthAverage:=HGW_Average_0.AverageLength;
	END_IF

(* Update Drawroll Gearing Based On Average Length *)
	IF (HGW_Average_0.Update) THEN
		gA[5].Cmd_SynchronizedMotionUpdate:=1;
		gReg[5].SP_Repeat:=HGW_Average_0.AverageLength;
	END_IF

(* Detect Change In Repeat Setpoint *)
	IF (gRecipeActive.Repeat<>Repeat_Old) THEN
		Repeat_Old:=gRecipeActive.Repeat;
		gA[5].Cmd_SynchronizedMotionUpdate:=1;
		gReg[5].SP_Repeat:=gRecipeActive.Repeat;
		gReg[5].LengthAverage:=gRecipeActive.Repeat;
		gReg[5].LengthActual:=gRecipeActive.Repeat;
		gReg[5].Enable:=0;
	END_IF
(* Detect Change In Drawroll Diameter Setpoint *)
	IF (gSP_A[5].Diameter<>Diameter_Old) THEN
		Diameter_Old:=gSP_A[5].Diameter;
		gA[5].Cmd_SynchronizedMotionUpdate:=1;
		gReg[5].Enable:=0;
	END_IF
(* Detect Change In Drawroll Format Setpoint *)
	IF (gReg[5].SP_Format<>Format_Old) THEN
		Format_Old:=gReg[5].SP_Format;
		gA[5].Cmd_SynchronizedMotionUpdate:=1;
		gReg[5].Enable:=0;
	END_IF
	IF (NOT gA[5].Ind_SynchronizedMotion) THEN
		gA[5].Cmd_SynchronizedMotionUpdate:=0;
	END_IF

(**** MISSED MARK SHUTDOWN SECTION ****)

(* Missed Mark Shutdown Count *)
	IF (gReg[5].SP_MarkMissedCount>0) THEN
		IF (gReg[5].MarkMissedNew) THEN
			MissedMark_Count:=MissedMark_Count+1;
			FirstAverage:=0;
		END_IF
	END_IF
  IF (gReg[5].MarkGoodNew OR NOT(gReg[5].Enable) OR gHMI_Reset_PB OR EDGEPOS(gQ_CR_EstopReset)) THEN
		MissedMark_Count:=0;
	END_IF

(* Missed Mark Shutdown Evaluation *)
	IF(MissedMark_Count>gReg[5].SP_MarkMissedCount) THEN
		gReg[5].ShutdownMissedMark:=1;
	ELSE
		gReg[5].ShutdownMissedMark:=0;
	END_IF

(**** REGISTRATION USER OFFSET WATCH ****)

(* Detect Change In User Offset *)
	IF (gReg[5].SP_Offset<>Offset_Old) THEN
		Offset_Old:=gReg[5].SP_Offset;
		IF (gReg[5].MarkFirst) THEN
			gReg[5].OffsetActive:=1;
		END_IF
	END_IF
(* Watch for 2 consecutive corrections < maximum...this will indicate the user offset is run in *)
	IF (gReg[5].OffsetActive=1) THEN
		IF ((gReg[5].MarkGoodNew)AND(NOT gReg[5].CorrectionMax)) THEN
			Count:=Count+1;
		END_IF
		IF ((Count>2)OR(NOT gReg[5].Enable)) THEN
			Count:=0;
			gReg[5].OffsetActive:=0;
		END_IF
	END_IF

(**** REGISTRATION OUT OF TOLERANCE SHUTDOWN SECTION ****)

(* Out Of Tolerance Shutdown Count *)
	IF (gReg[5].SP_OutOfToleranceCount>0) THEN
		IF (gReg[5].MarkGoodNew) THEN
			IF ((gReg[5].CorrectionMax)AND(NOT gReg[5].OffsetActive)) THEN
				OutOfTolerance_Count:=OutOfTolerance_Count+1;
			ELSE
			OutOfTolerance_Count:=0;
			END_IF
		END_IF
	END_IF
	IF ((NOT gReg[5].Enable) OR gHMI_Reset_PB) THEN
		OutOfTolerance_Count:=0;
	END_IF

(* Out Of Tolerance Shutdown Evaluation *)
	IF (OutOfTolerance_Count>gReg[5].SP_OutOfToleranceCount) THEN
		gReg[5].ShutdownOutOfTolerance:=1;
	ELSE
		gReg[5].ShutdownOutOfTolerance:=0;
	END_IF

	(* General Reset Of Notification Bools *)
	gReg[5].MarkMissedNew:=0;
	gReg[5].MarkGoodNew:=0;
	gReg[5].CorrectionMax:=0;

END_PROGRAM
```

### Program Logical/BagMachine_Section/EnvBag/Axis12/A12_Automat (IEC)

#### A12_AutomatCyclic.st - Cyclic code
```iecst
(********************************************************************
 * COPYRIGHT -- Microsoft
 ********************************************************************
 * Program: A12_Automat
 * File: A12_AutomatCyclic.st
 * Author: dominique
 * Created: November 21, 2011
 ********************************************************************
 * Implementation of program A12_Automat
 ********************************************************************)

PROGRAM _CYCLIC

    // Synchro ratio Master/Slave
    iIndex := MC_BR_AutControl_0.ActualStateIndex ;
    IF gRecipeActive.bSelEnvBProd THEN
      CASE iIndex OF
        3 : // Master = Tearing
           //gA[12].rRSynNum := 1.0 ;         D.M. 03/02/2012 Pyrollpack_14661 Suppress cause is not correct for offset Virtual Masrter / Slave calculation in A4_Basic and not used in setting mode Automat state 3
           //gA[12].rRSynDen := 2.0 ;
      ELSE  // Master = Virtual
           //gA[12].rRSynNum := 1.0 ;
           //gA[12].rRSynDen := 1.0 ;
      END_CASE
      // Master = Virtual
      gA[12].rRSynNum := 1.0 ;
      gA[12].rRSynDen := 1.0 ;
    ELSE
      CASE iIndex OF
        3 : // Master = Tearing
           //gA[12].rRSynNum := 1.0 ;
           //gA[12].rRSynDen := 4.0 ;
      ELSE  // Master = Virtual
           IF (g_rNumbPliers <> 0.0) THEN
             gA[12].rRSynDen := g_rNumbPliers ;
           ELSE
             gA[12].rRSynDen := 4.0 ;
           END_IF
           gA[12].rRSynNum := 1.0 ;
      END_CASE
    END_IF

(**** STRAIGHT GEARED CAM AUTOMAT WITH ABSOLUTE PHASE SYNCHRONIZATION FOR ENVELOPE BAG AXIS ***)

(* Set Up Master Position Parameter ID *)

  // Holding+Tearing+EnvBag+TearEB+Drum timing setting
  IF gstCycA[3].CycManTimSet.CmdSynchroOn OR
     gstCycA[4].CycManTimSet.CmdSynchroOn THEN
    MC_BR_AutControl_0.Signal1 := 1 ;
    MC_BR_AutControl_0.Signal2 := 0 ;
  ELSE
    MC_BR_AutControl_0.Signal1 := 0 ;
    MC_BR_AutControl_0.Signal2 := 1 ;
  END_IF

  // A12 Synchro OK indicator
  gstCycA[3].CycManTimSet.bSynchroOkSlavA[12] := ( MC_BR_InitMasterParIDTransfer_1.Master = gA[4].Ident )                                AND
                                                 ( MC_BR_InitMasterParIDTransfer_1.MasterParID = gstCycA[4].CycManTimSet.uiMasterParID ) AND
                                                 ( MC_BR_AutControl_0.ActualStateIndex = 3 )                                             AND
                                                 gA[12].Ind_SynchronizedMotion AND ParID_Ready ;

  // A12 Synchro OK indicator
  gstCycA[4].CycManTimSet.bSynchroOkSlavA[12] := ( MC_BR_InitMasterParIDTransfer_1.Master = gA[4].Ident )                                AND
                                                 ( MC_BR_InitMasterParIDTransfer_1.MasterParID = gstCycA[4].CycManTimSet.uiMasterParID ) AND
                                                 ( MC_BR_AutControl_0.ActualStateIndex = 3 )                                             AND
                                                 gA[12].Ind_SynchronizedMotion AND ParID_Ready ;

  // EnvBag+TearEB+Drum timing setting
  IF gstCycA[12].CycManTimSet.bCyc THEN
    IF (gstCycA[12].CycManTimSet.CmdSynchroOn) THEN
      MC_BR_AutControl_0.Signal1 := 0 ;
      MC_BR_AutControl_0.Signal2 := 0 ;
      MC_BR_AutControl_0.Signal3 := 1 ;
    ELSE
      MC_BR_AutControl_0.Signal1 := 0 ;
      MC_BR_AutControl_0.Signal2 := 0 ;
      MC_BR_AutControl_0.Signal3 := 0 ;
    END_IF
  END_IF

  // A12 Synchro OK indicator
  gstCycA[12].CycManTimSet.bSynchroOkSlavA[12] := ( MC_BR_AutControl_0.ActualStateIndex = 2 )   AND
                                                  gA[12].Ind_SynchronizedMotion AND ParID_Ready ;

  IF gstCycA[3].CycManTimSet.bFCyc  AND
     gstCycA[4].CycManTimSet.bFCyc  AND
     gstCycA[12].CycManTimSet.bFCyc THEN
    MC_BR_AutControl_0.Signal1 := 0 ;
    MC_BR_AutControl_0.Signal2 := 0 ;
    MC_BR_AutControl_0.Signal3 := 0 ;
  END_IF

  // Slave Period
  IF gRecipeActive.bSelEnvBProd THEN
    rSlave_TimingAxisPeriod := gA[12].AxisPeriod / 2.0 ; // Tearing Axis is Master
    rSlave_AxisPeriod       := gA[12].AxisPeriod ;       // Virtual Master Axis is Master
  ELSE
    rSlave_TimingAxisPeriod := gA[12].AxisPeriod / 4.0 ; // Tearing Axis is Master
    rSlave_AxisPeriod       := gA[12].AxisPeriod / g_rNumbPliers ; // Virtual Master Axis is Master
  END_IF

  //Synch_Request := gA[12].Cmd_SynchronizedMotion ;
  Synch_Request := gA[12].Cmd_SynchronizedMotion AND NOT(MC_BR_AutControl_0.Stop) ;  // D.M. 26/01/2012 RS26 Pyrollpack_14661 added because it happened that Stop=1 and Synch_Request=1 => MC_BR_AutControl_0 makes fault 29256
	IF (Synch_Request AND NOT ParID_Ready) THEN
    MC_BR_InitMasterParIDTransfer_0.Master:= gA[9].Ident ;
    MC_BR_InitMasterParIDTransfer_0.Slave:=gA[12].Ident;
    MC_BR_InitMasterParIDTransfer_0.MasterParID:= 412 ; // ParID 412 = VAX Position (in case virtual axis)
    MC_BR_InitMasterParIDTransfer_0.SlaveChannel:=0;
    MC_BR_InitMasterParIDTransfer_0.Execute:= 1 ;
    IF (MC_BR_InitMasterParIDTransfer_0.Done) THEN
      MasterParID:=MC_BR_InitMasterParIDTransfer_0.ReceiveParID;
      MC_BR_InitMasterParIDTransfer_0.Execute:=FALSE;
      ParID_Ready1:=1;
    ELSIF (MC_BR_InitMasterParIDTransfer_0.Error) THEN
    (*Store ErrorID in a variable,
      ErrorID is reset on falling edge of 'Execute'*)
      ErrorID:=MC_BR_InitMasterParIDTransfer_0.ErrorID;
      ParID_Ready1:=0;
      MC_BR_InitMasterParIDTransfer_0.Execute:=FALSE;
    END_IF
    MC_BR_InitMasterParIDTransfer_1.Master       := gA[4].Ident ;
    MC_BR_InitMasterParIDTransfer_1.Slave        := gA[12].Ident;
    MC_BR_InitMasterParIDTransfer_1.MasterParID  := gstCycA[12].CycManTimSet.uiMasterParID ;
    MC_BR_InitMasterParIDTransfer_1.SlaveChannel := 2 ;
    MC_BR_InitMasterParIDTransfer_1.Execute      := 1 ;
    IF (MC_BR_InitMasterParIDTransfer_1.Done) AND ParID_Ready1 THEN
      uiMasterParID1:=MC_BR_InitMasterParIDTransfer_1.ReceiveParID;
      MC_BR_InitMasterParIDTransfer_1.Execute:=FALSE;
      ParID_Ready:=1;
    ELSIF (MC_BR_InitMasterParIDTransfer_1.Error) THEN
    (*Store ErrorID in a variable,
      ErrorID is reset on falling edge of 'Execute'*)
      ErrorID:=MC_BR_InitMasterParIDTransfer_1.ErrorID;
      ParID_Ready:=0;
      MC_BR_InitMasterParIDTransfer_1.Execute:=FALSE;
    END_IF
	END_IF
  MC_BR_InitMasterParIDTransfer_0();
  MC_BR_InitMasterParIDTransfer_1();

(**** Initialize Automat Parameters Upon Automat Start Request ****)
	IF (EDGEPOS(ParID_Ready))THEN

		//*** Calculate Slave Start Offset ****
			MasterOffset := gRecipeActive.Tearing_Offset+gRecipeActive.Holding_Offset;
			PositionOffset:= REAL_TO_DINT((gA[9].PositionInch-(gA[12].PositionInch-MasterOffset))*1000);
			PositionMOD:= REAL_TO_DINT(gRecipeActive.Repeat*1000);
			SlaveStartOffset:= (DINT_TO_REAL(PositionOffset MOD PositionMOD))/1000;
			IF (SlaveStartOffset >= (0.5*gRecipeActive.Repeat)) THEN
				SlaveStartOffset := SlaveStartOffset - gRecipeActive.Repeat;
			END_IF
			IF (SlaveStartOffset < (-0.5*gRecipeActive.Repeat)) THEN
				SlaveStartOffset := SlaveStartOffset + gRecipeActive.Repeat;
			END_IF

      IF gRecipeActive.bSelEnvBProd AND
         gr_rIndEnvB2AxTear1        AND
         1                          THEN
        // Mecanic ratio between EnvB Axis and Lower roller of Envelope Bag Station = 45/30 = 3/2
        // Lower Roller Envelope Bag Station performs 2 revolutions per bag to come back on the same position for each bag and run faster than tearing belts carriage to not obstruct the bag way
        rSlave_AxisPeriod := 2 * 2/3 * gA[12].AxisPeriod ;
      ELSE
        rSlave_AxisPeriod := gA[12].AxisPeriod * gA[12].rRSynNum/gA[12].rRSynDen ;
      END_IF
      rOffsetDeg := gRecipeActive.rEnvB_PhasMasterDeg ;

      rSPMaPos := (gA[12].PositionDeg - rOffsetDeg)/(gA[12].rRSynNum/gA[12].rRSynDen) ;
      rTemp_[1] := gA[12].PositionDeg ;
      rTemp_[0] := rSPMaPos - gA[9].PositionDeg ;
      rMaCompDist := H_FC_Modulus (
                          //IN_rMod := (360 * gA[12].rRSynNum/gA[12].rRSynDen) ,
                          IN_rMod := 360 ,
                          IN_rVar := rTemp_[0]
                                  ) ;

		(*general automat parameter*)
			//AutData.Master				    := gA[3].Ident;
			AutData.MasterParID			  := MasterParID;
			AutData.StartPosition		  := 0;
			AutData.StartInterval		  := gA[9].AxisPeriod;
			AutData.MaxMasterVelocity	:= gr_rMachMaxSpeed_BPM ;

		//Automat STATE 0 Basis State
			AutData.State[0].Event[0].Type		  := ncST_END;
			AutData.State[0].Event[0].Attribute	:= ncAT_ONCE;
      IF (rMaCompDist >= 1/gA[9].UnitsPerDeg) AND // rMaCompDist must be >= 1 Units
         gA[12].bSynchroReq                   THEN
		  	AutData.State[0].Event[0].NextState	:= 1;
      ELSE
        rMaCompDist := 1/gA[9].UnitsPerDeg ;
        AutData.State[0].Event[0].NextState := 2;
      END_IF

    //Automat STATE 1 Master/Slave Absolute Phase Correction
      AutData.State[1].MasterParID        := MasterParID;
      AutData.State[1].CamProfileIndex    := 16#FFFF;
      AutData.State[1].MasterFactor       := REAL_TO_UDINT(rMaCompDist * gA[12].UnitsPerDeg) ;
      AutData.State[1].SlaveFactor        := 0 ;
      AutData.State[1].CompMode           := ncOFF;

      AutData.State[1].Event[0].Type      := ncST_END ;
      AutData.State[1].Event[0].Attribute := ncST_END ;
      AutData.State[1].Event[0].NextState := 2 ;

      AutData.State[1].Event[1].Type      := ncSIGNAL1 ;
      AutData.State[1].Event[1].Attribute := ncAT_ONCE ;
      AutData.State[1].Event[1].NextState := 3 ;

      AutData.State[1].Event[2].Type      := ncSIGNAL3 ;
      AutData.State[1].Event[2].Attribute := ncAT_ONCE ;
      AutData.State[1].Event[2].NextState := 2 ;

    //Automat STATE 2 Master/Slave run
      AutData.State[2].MasterParID     := MasterParID;
      AutData.State[2].CamProfileIndex := 16#FFFF;
      AutData.State[2].MasterFactor    := REAL_TO_UDINT(gA[9].AxisPeriod);
      AutData.State[2].SlaveFactor     := REAL_TO_UDINT(rSlave_AxisPeriod);
      AutData.State[2].CompMode        := ncOFF;

      AutData.State[2].Event[0].Type      := ncST_END ;
      AutData.State[2].Event[0].Attribute := ncST_END;
      AutData.State[2].Event[0].NextState := 2;

      AutData.State[2].Event[1].Type      := ncST_END+ncNEGATIVE ;
      AutData.State[2].Event[1].Attribute := ncST_END;
      AutData.State[2].Event[1].NextState := 2;

      AutData.State[2].Event[2].Type      := ncSIGNAL1;
      AutData.State[2].Event[2].Attribute := ncAT_ONCE;
      AutData.State[2].Event[2].NextState := 3;

    //Automat STATE 3 Master/Slave Timing setting
      AutData.State[3].MasterParID     := uiMasterParID1;
      AutData.State[3].CamProfileIndex := 16#FFFF;
      AutData.State[3].MasterFactor    := REAL_TO_UDINT(gA[4].AxisPeriod);
      AutData.State[3].SlaveFactor     := REAL_TO_UDINT(rSlave_TimingAxisPeriod);
      AutData.State[3].CompMode        := ncOFF;

      AutData.State[3].Event[0].Type       := ncST_END ;
      AutData.State[3].Event[0].Attribute  := ncST_END ;
      AutData.State[3].Event[0].NextState  := 3 ;

      AutData.State[3].Event[1].Type       := ncST_END+ncNEGATIVE ;
      AutData.State[3].Event[1].Attribute  := ncST_END ;
      AutData.State[3].Event[1].NextState  := 3 ;

      AutData.State[3].Event[2].Type       := ncSIGNAL2 ;
      AutData.State[3].Event[2].Attribute  := ncAT_ONCE ;
      AutData.State[3].Event[2].NextState  := 2 ;

      MC_BR_AutControl_0.Enable      := 1;
      MC_BR_AutControl_0.AdrAutData  := ADR(AutData);
      MC_BR_AutControl_0.InitAutData := 1;
  END_IF

			(* wait for initialization done or restart *)
			IF ((MC_BR_AutControl_0.AutDataInitialized=1) AND (Synch_Request)) THEN
				MC_BR_AutControl_0.InitAutData := 0;
				MC_BR_AutControl_0.Enable :=1;
				AutomatStart := 1;
        uiMC_BR_AutControl_0_MemoErrorID := 0 ;
			END_IF
			(* check if error occured *)
			IF (MC_BR_AutControl_0.ErrorID <> 0) THEN
        uiMC_BR_AutControl_0_MemoErrorID := MC_BR_AutControl_0.ErrorID ;
				MC_BR_AutControl_0.Enable := 0;
			END_IF

	(******************** ENABLE CAM-AUTOMAT **********************)

	IF (AutomatStart) THEN
			MC_BR_AutControl_0.Start := 1;
			AutomatStart := 0;
	END_IF

	IF (NOT Synch_Request) THEN
			MC_BR_AutControl_0.Stop := 1;
			MC_BR_AutControl_0.Start := 0;
      ParID_Ready := 0;
      ParID_Ready1 := 0;
			IF (MC_BR_AutControl_0.Running=0) THEN
				MC_BR_AutControl_0.Enable := 0;
				MC_BR_AutControl_0.Stop := 0;
        g_bEnvBagSelectChang := 0 ;
			END_IF
   //*************************************************
   // D.M. 26/01/2012 RS26 Pyrollpack_14661 added because after guard fault it happened that Stop=1 and MC_BR_AutControl_0.Enable => not possible to finish MC_BR_AutControl_0 => program locked
      IF MC_BR_AutControl_0.Stop        AND
         NOT(MC_BR_AutControl_0.Enable) THEN
        MC_BR_AutControl_0.Enable := 1 ;
      END_IF
   //*************************************************
  END_IF

	gA[12].Ind_AutomatEnabled:=MC_BR_AutControl_0.Enable;
	gA[12].Ind_CurrentAutomatState:=MC_BR_AutControl_0.ActualStateIndex;
  gA[12].Ind_bSynchroOK := (MC_BR_AutControl_0.ActualStateIndex >= 2) AND gA[12].Ind_SynchronizedMotion ; ;

	(********************** MC_AUTCONTROL *************************)
	MC_BR_AutControl_0.Slave:= gA[12].Ident;
	MC_BR_AutControl_0();

(******************** UPDATE CAM-AUTOMAT STATE 2 **********************)
  IF g_bEnvBagSelectChang                      AND
     (MC_BR_AutControl_0.ActualStateIndex = 2) THEN
    MC_BR_InitAutState_0.Execute := 1 ;
    uiInitAutState_0_MemoErrorID := 0 ;
  END_IF
  MC_BR_InitAutState_0.MasterParID     := MasterParID ;
  MC_BR_InitAutState_0.Slave           := gA[12].Ident ;
  MC_BR_InitAutState_0.StateIndex      := 2 ;
  MC_BR_InitAutState_0.CamProfileIndex := 16#FFFF ;
  MC_BR_InitAutState_0.MasterFactor    := REAL_TO_UDINT(gA[9].AxisPeriod) ;
  MC_BR_InitAutState_0.SlaveFactor     := REAL_TO_DINT(rSlave_AxisPeriod) ;
  MC_BR_InitAutState_0.CompMode        := ncOFF ;
  MC_BR_InitAutState_0() ;

  IF (MC_BR_InitAutState_0.Done)  OR
     (MC_BR_InitAutState_0.Error) THEN
    MC_BR_InitAutState_0.Execute := 0;
    uiInitAutState_0_MemoErrorID := MC_BR_InitAutState_0.ErrorID ;
  END_IF

END_PROGRAM
```

#### A12_Automat.var - Local variables
```iecst
(********************************************************************
 * COPYRIGHT -- Microsoft
 ********************************************************************
 * Program: A12_Automat
 * File: A12_Automat.var
 * Author: dominique
 * Created: November 21, 2011
 ********************************************************************
 * Local variables of program A12_Automat
 ********************************************************************)
VAR
	AutData : MC_AUTDATA_TYP;
	AutomatStart : BOOL;
	ErrorID : UINT;
	MasterOffset : REAL;
  MasterParID : UINT;
  uiMasterParID1 : UINT;
  uiSP_MasterParID : UINT;
  uiiSP_Master : UDINT;
  bCmdSynchroOn : BOOL ;
  bCmdSynchroOff : BOOL ;
  bCmdSynchroOn1 : BOOL ;
  bCmdSynchroOff1 : BOOL ;
  uiiSP_MasterFactor : UDINT ;
  uiiSP_SlaveFactor : UDINT ;
	MC_BR_AutControl_0 : MC_BR_AutControl;
  uiMC_BR_AutControl_0_MemoErrorID : UINT ;
  MC_BR_InitMasterParIDTransfer_0 : MC_BR_InitMasterParIDTransfer;
  MC_BR_InitMasterParIDTransfer_1 : MC_BR_InitMasterParIDTransfer;
  ParID_Ready : BOOL;
  ParID_Ready1 : BOOL;
	PositionMOD : DINT;
	PositionOffset : DINT;
	SlaveStartOffset : REAL;
	Synch_Request : BOOL;
  bTest_ : ARRAY[0..9] OF  BOOL;
  iTest_ : ARRAY[0..9] OF  INT;
  rTest_ : ARRAY[0..9] OF  REAL;
  rMaCompDist : REAL ;
  rSPMaPos    : REAL ;
  rOffsetDeg  : REAL ;
  rSlCompDist : REAL ;
  rTemp_      : ARRAY[0..9] OF REAL ;
  usiMemoStat : USINT;
  iIndex : INT ;
  rMaCompDistStat6 : REAL;
  rSlCompDistStat6 : REAL;
  rMasterFactor5 : REAL;
  iiMasterFactor5 : DINT;
  iiSlaveFactor5  : DINT;
  rSlave_AxisPeriod : REAL ;
  rSlave_TimingAxisPeriod : REAL ;
  MC_BR_InitAutState_0 : MC_BR_InitAutState;
  uiInitAutState_0_MemoErrorID : UINT ;
END_VAR
```

### Program Logical/BagMachine_Section/EnvBag/Axis12/A12_Control (IEC)

#### A12_ControlCyclic.ld - Cyclic code
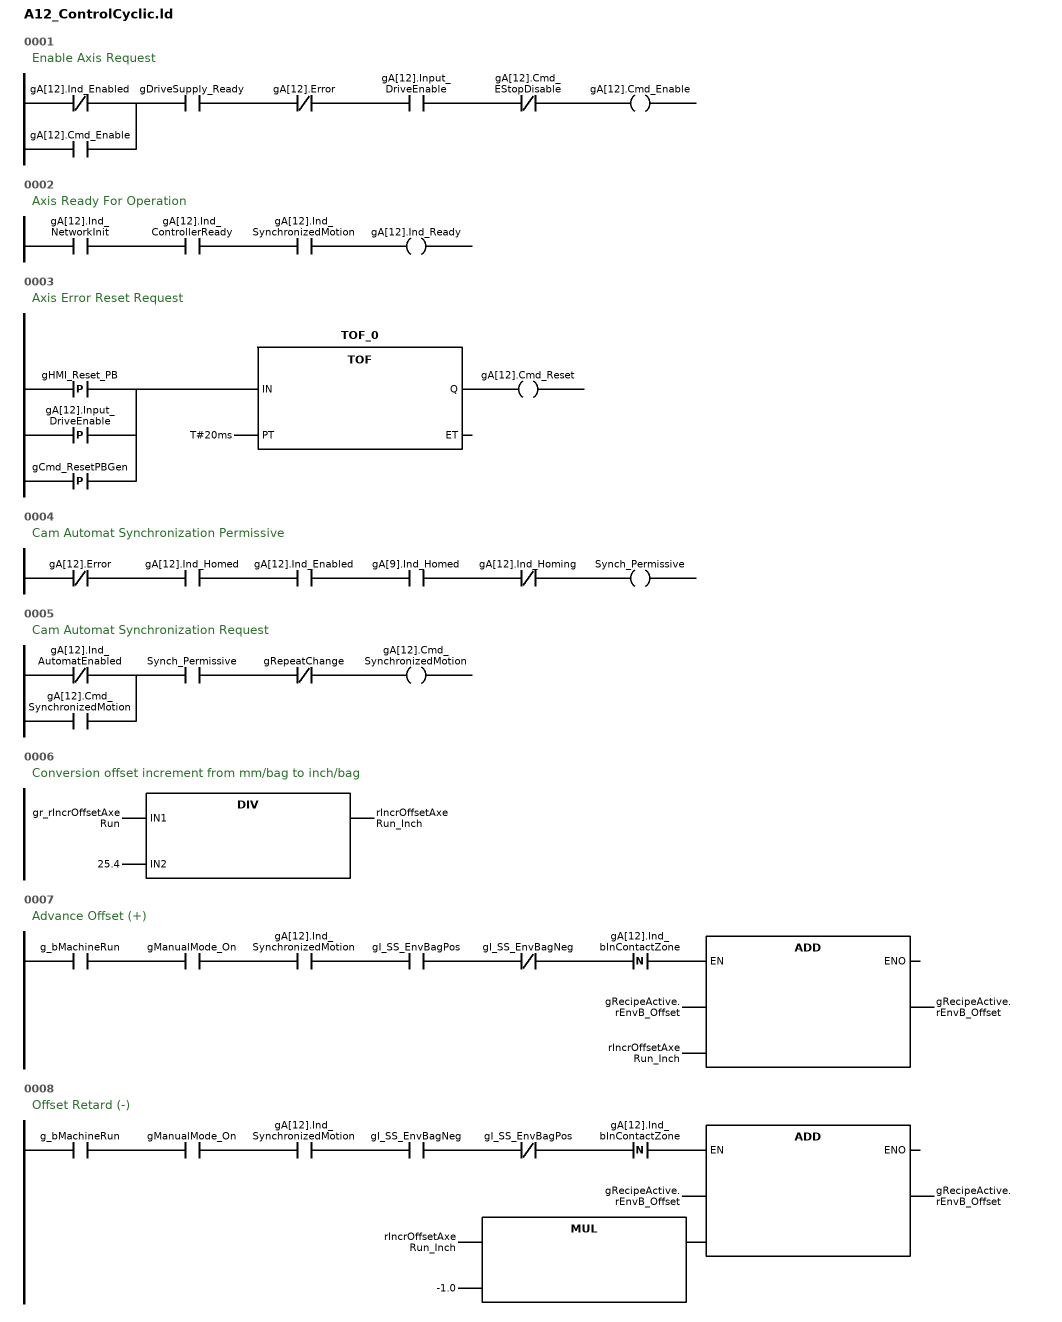
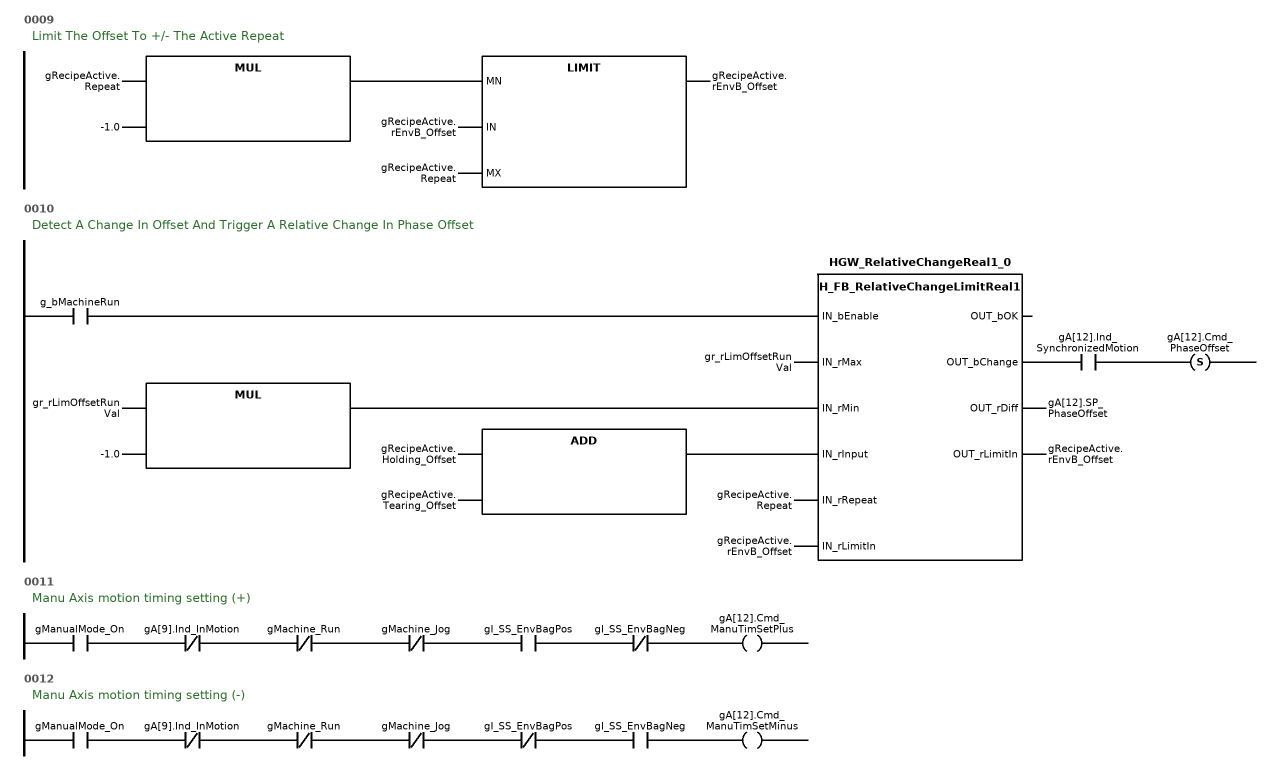
Ladder, written as Structured Text:
```iecst
(********************************************************************
 * COPYRIGHT -- Microsoft
 ********************************************************************
 * Program: A4_Control
 * File: A4_ControlCyclic.ld
 * Author: pkiel
 * Created: July 13, 2011
 ********************************************************************
 * Implementation of program A4_Control
 ********************************************************************)

PROGRAM _CYCLIC
VAR
    _e1 : R_TRIG;
    _e2 : R_TRIG;
    _e3 : R_TRIG;
    _e4 : F_TRIG;
    _e5 : F_TRIG;
END_VAR
(* Network 1: Enable Axis Request *)
gA[12].Cmd_Enable := (NOT gA[12].Ind_Enabled OR gA[12].Cmd_Enable) AND gDriveSupply_Ready AND NOT gA[12].Error AND gA[12].Input_DriveEnable AND NOT gA[12].Cmd_EStopDisable;

(* Network 2: Axis Ready For Operation *)
gA[12].Ind_Ready := gA[12].Ind_NetworkInit AND gA[12].Ind_ControllerReady AND gA[12].Ind_SynchronizedMotion;

(* Network 3: Axis Error Reset Request *)
_e1(CLK := gHMI_Reset_PB);
_e2(CLK := gA[12].Input_DriveEnable);
_e3(CLK := gCmd_ResetPBGen);
TOF_0(IN := _e1.Q OR _e2.Q OR _e3.Q, PT := T#20ms);
gA[12].Cmd_Reset := TOF_0.Q;

(* Network 4: Cam Automat Synchronization Permissive *)
Synch_Permissive := NOT gA[12].Error AND gA[12].Ind_Homed AND gA[12].Ind_Enabled AND gA[9].Ind_Homed AND NOT gA[12].Ind_Homing;

(* Network 5: Cam Automat Synchronization Request *)
gA[12].Cmd_SynchronizedMotion := (NOT gA[12].Ind_AutomatEnabled OR gA[12].Cmd_SynchronizedMotion) AND Synch_Permissive AND NOT gRepeatChange;

(* Network 6: Conversion offset increment from mm/bag to inch/bag *)
rIncrOffsetAxeRun_Inch := gr_rIncrOffsetAxeRun / 25.4;

(* Network 7: Advance Offset (+) *)
_e4(CLK := gA[12].Ind_bInContactZone);
IF g_bMachineRun AND gManualMode_On AND gA[12].Ind_SynchronizedMotion AND gI_SS_EnvBagPos AND NOT gI_SS_EnvBagNeg AND _e4.Q THEN
    gRecipeActive.rEnvB_Offset := gRecipeActive.rEnvB_Offset + rIncrOffsetAxeRun_Inch;
END_IF;

(* Network 8: Offset Retard (-) *)
_e5(CLK := gA[12].Ind_bInContactZone);
IF g_bMachineRun AND gManualMode_On AND gA[12].Ind_SynchronizedMotion AND gI_SS_EnvBagNeg AND NOT gI_SS_EnvBagPos AND _e5.Q THEN
    gRecipeActive.rEnvB_Offset := gRecipeActive.rEnvB_Offset + (rIncrOffsetAxeRun_Inch * -1.0);
END_IF;

(* Network 9: Limit The Offset To +/- The Active Repeat *)
gRecipeActive.rEnvB_Offset := LIMIT(MN := gRecipeActive.Repeat * -1.0, IN := gRecipeActive.rEnvB_Offset, MX := gRecipeActive.Repeat);

(* Network 10: Detect A Change In Offset And Trigger A Relative Change In Phase Offset *)
HGW_RelativeChangeReal1_0(IN_bEnable := g_bMachineRun, IN_rMax := gr_rLimOffsetRunVal, IN_rMin := gr_rLimOffsetRunVal * -1.0, IN_rInput := gRecipeActive.Holding_Offset + gRecipeActive.Tearing_Offset, IN_rRepeat := gRecipeActive.Repeat, IN_rLimitIn := gRecipeActive.rEnvB_Offset);
IF HGW_RelativeChangeReal1_0.OUT_bChange AND gA[12].Ind_SynchronizedMotion THEN
    gA[12].Cmd_PhaseOffset := TRUE;
END_IF;
gA[12].SP_PhaseOffset := HGW_RelativeChangeReal1_0.OUT_rDiff;
gRecipeActive.rEnvB_Offset := HGW_RelativeChangeReal1_0.OUT_rLimitIn;

(* Network 11: Manu Axis motion timing setting (+) *)
gA[12].Cmd_ManuTimSetPlus := gManualMode_On AND NOT gA[9].Ind_InMotion AND NOT gMachine_Run AND NOT gMachine_Jog AND gI_SS_EnvBagPos AND NOT gI_SS_EnvBagNeg;

(* Network 12: Manu Axis motion timing setting (-) *)
gA[12].Cmd_ManuTimSetMinus := gManualMode_On AND NOT gA[9].Ind_InMotion AND NOT gMachine_Run AND NOT gMachine_Jog AND NOT gI_SS_EnvBagPos AND gI_SS_EnvBagNeg;
END_PROGRAM
```

### Program Logical/BagMachine_Section/EnvBag/Axis12/A12_Cycle
